// TwinCAT 3 PLC project Robotic
// ProgramVersion: 3.1.4023.0
// libraries:
//   CmpBitmapPool, * (System)
//   VisuElemMeter, * (System)
//   Tc2_EtherCAT, * (Beckhoff Automation GmbH)
//   Tc2_Standard, * (Beckhoff Automation GmbH)
//   Tc2_SUPS, * (Beckhoff Automation GmbH)
//   Tc2_System, * (Beckhoff Automation GmbH)
//   Tc2_Utilities, * (Beckhoff Automation GmbH)
//   Tc3_Module, * (Beckhoff Automation GmbH)
//   VisuDialogs, * (System)
//   VisuSymbols,3.5.10.0,System
//   VLT_ECAT_LIB_V1_12,1.12,Danfoss Drives
// project tree:
//   DUTs/OEE/ ShiftTime.TcDUT, Precentage_Time.TcDUT, ShiftCounter.TcDUT, sOEECounter.TcDUT, StartShift_EndShift.TcDUT, sOEETime.TcDUT
//   DUTs/Robot/ stCustomPattern.TcDUT, stProductInfo.TcDUT, stRobot_Input.TcDUT, stRobot_Output.TcDUT, unMyINT.TcDUT, unMyUINT.TcDUT
//   DUTs/ stCheckShuttle.TcDUT, stDM_Input.TcDUT, stDM_Output.TcDUT, stEcSlaveState.TcDUT, stErrorData.TcDUT, stMachineState.TcDUT, stMotor.TcDUT, stPalletTrackingData.TcDUT, stPneumatic1.TcDUT, stPneumatic2.TcDUT, stRejectData.TcDUT, stRTC_Data.TcDUT, stShuttle.TcDUT, stDataPallet.TcDUT
//   / Ethernet_Task.TcTTO, GlobalTextList.TcGTLO, IO_Task.TcTTO, Main_Task.TcTTO, Monitoring_Task.TcTTO, VISU_TASK.TcTTO
//   GVLs/ Data_GVL.TcGVL, HMI_GVL.TcGVL, InputOutput_GVL.TcGVL, Status_GVL.TcGVL
//   POUs/Function/ ConvertMilliSecTimeData.TcPOU, ConvertTimeToString.TcPOU
//   POUs/Function_Block/ FB_CheckShuttlePos.TcPOU
//   POUs/Function_Block/General/ Alarm_Event_History.TcPOU, Alarm_Event_Active.TcPOU, BLINK.TcPOU, CheckStatus.TcPOU, Ethercat_Status.TcPOU, FB_StateManager.TcPOU, FGHS_DataCollect_Palletizing.TcPOU, MotorManagement.TcPOU, OEETime.TcPOU, OEECounter.TcPOU, Pneumatic_1Coil_Management.TcPOU, Pneumatic_2Coil_Management.TcPOU, RejectMsgHandling.TcPOU, RTCManagement.TcPOU, SystemData.TcPOU
//   POUs/Function_Block/Placing/ FB_CustomOffset.TcPOU, FB_Placing.TcPOU, FB_Placing_v2.TcPOU, PalletID_Name.TcPOU
//   POUs/Function_Block/Robot/ DM_Connect.TcPOU, FB_BarcodeInspection.TcPOU, FB_Picking.TcPOU, FB_Recipe.TcPOU, RobotCustomPattern.TcPOU, FB_StartUpRobot.TcPOU, FB_Layer.TcPOU, RotatePick.TcPOU
//   POUs/S00_System_Utilities/ Backbone.TcPOU, IO_Mapping.TcPOU, Module_Status.TcPOU
//   POUs/S01_Robot/ EM01_Robot.TcPOU, EM06_Picking.TcPOU
//   POUs/S02_Placing/ EM02_Placing1.TcPOU, EM03_Placing2.TcPOU, EM04_Placing3.TcPOU, EM05_Placing4.TcPOU
//   VISUs/FGHS/ DataPallet2.TcVIS, DataPallet3.TcVIS, DataPallet4.TcVIS, FGHS.TcVIS, FGHS_1.TcVIS, DataPallet1.TcVIS
//   VISUs/Images/ ImagePool.TcIPO (not stored)
//   VISUs/Main/Alarm/ RejectMsg.TcVIS, AlarmHistory.TcVIS, AlarmActive.TcVIS, Alarm.TcVIS, PUDetail.TcVIS
//   VISUs/Main/ Header.TcVIS, Home.TcVIS, MainPage.TcVIS, Parameter.TcVIS, PLC_Status.TcVIS, PUSeq.TcVIS, StateMachine.TcVIS
//   VISUs/MTBF/ MTBF.TcVIS, MTBF_Picking.TcVIS, MTBF_Placing.TcVIS, MTBF_Outfeed.TcVIS, MTBF_Infeed.TcVIS, MTBF_Shuttle.TcVIS, MTBF_Dispenser.TcVIS
//   VISUs/OEE/ OEE.TcVIS, OEE_Outfeed.TcVIS, OEE_Robot.TcVIS, OEE_Counter.TcVIS
//   VISUs/Parameter/ LinkUp.TcTLO, MShuttle.TcVIS, MOutfeed.TcVIS, MInfeed.TcVIS, MDispenser.TcVIS, MPicking.TcVIS, MPlacing.TcVIS
//   VISUs/Parameter/Recipe/ MOffset_2.TcVIS, MOffset_3.TcVIS, MOffset_4.TcVIS, MRecipe.TcVIS, MRecipe_1.TcVIS, MOffset_1.TcVIS, MRecipe_2.TcVIS, MRecipe_3.TcVIS, MRecipe_4.TcVIS
//   VISUs/PLC Status/P1 - Panel Robot/ P1_DI1.TcVIS, P1_DI2.TcVIS, P1_DI3.TcVIS, P1_DI4.TcVIS, P1_DO1.TcVIS, P1_DO2.TcVIS, P1_DO3.TcVIS
//   VISUs/PLC Status/P2 - Panel Outfeed/ P2_DI1.TcVIS, P2_DI2.TcVIS, P2_DI3.TcVIS, P2_DI4.TcVIS, P2_DI5.TcVIS, P2_DI6.TcVIS, P2_DI7.TcVIS, P2_DO1.TcVIS, P2_DO2.TcVIS, P2_DO3.TcVIS, P2_DO4.TcVIS
//   VISUs/PLC Status/P3 - Panel Shuttle/ P3_DI1.TcVIS, P3_DO1.TcVIS
//   VISUs/PLC Status/ SeqStatus.TcVIS, IO_Status.TcVIS
//   VISUs/TestMode/ Test_Outfeed.TcVIS, Control.TcVIS, Test_Infeed.TcVIS, Test_Place1.TcVIS, Test_Place2.TcVIS, Test_Place3.TcVIS, Test_Place4.TcVIS, Test_Shuttle.TcVIS, Test_Picking.TcVIS
//   VISUs/ VisualizationManager.TcVMO (not stored)
// real-time tasks:
//   TASK Main_Task: cycle T#4ms, priority 2, ADS port 350
//   TASK IO_Task: cycle T#2ms, priority 1, ADS port 351
//   TASK Monitoring_Task: cycle T#10ms, priority 10, ADS port 352
//   TASK Ethernet_Task: cycle T#100000us, priority 3, ADS port 353
//   TASK VISU_TASK: cycle T#100000us, priority 30, ADS port 354
// I/O:
//   DEVICE Main Panel (EtherCAT), AmsNetId 5.104.237.244.2.1
//     Term 1 (EK1200) [EK1200-5000 EtherCAT Power supply (2A E-Bus)]
//       Term 2 (EL1809) [EL1809 16Ch. Dig. Input 24V, 3ms]
//       Term 3 (EL1809) [EL1809 16Ch. Dig. Input 24V, 3ms]
//       Term 4 (EL1809) [EL1809 16Ch. Dig. Input 24V, 3ms]
//       Term 5 (EL1809) [EL1809 16Ch. Dig. Input 24V, 3ms]
//       Term 6 (EL2809) [EL2809 16Ch. Dig. Output 24V, 0.5A]
//       Term 7 (EL2809) [EL2809 16Ch. Dig. Output 24V, 0.5A]
//       Term 8 (EL2809) [EL2809 16Ch. Dig. Output 24V, 0.5A]
//       DeviceNet Master (EL6752) [EL6752 DeviceNet Master]
//   DEVICE Device 2 (EL6752), AmsNetId 5.104.237.244.3.1
//     Box 10 (Robot) // EDS-File: 'IRC5_Slave_DSQC1006.eds' DescText: Molex SST-DN4 Scanner EDS File Vendor: Molex Software & Electronics (SST) Device Type: Communication Adapter Product Name: Molex SST-DN4 Scanner Catalog Number: 0
//   DEVICE Ethernet/IP, AmsNetId 5.104.237.244.4.1
//     Box 11 (DataMan 300 Series Reader) // <INFO> </INFO> <EDS> C:\TwinCAT\3.1\Config\Io\EtherNetIP\0678077312900100.eds </EDS>
//     Box 12 (DataMan 260 Series Reader) (disabled) // <INFO> </INFO> <EDS> C:\TwinCAT\3.1\Config\Io\EtherNetIP\0678077313070100.eds </EDS>
//     Box 13 (DataMan 260 Series Reader) (disabled) // <INFO> </INFO> <EDS> C:\TwinCAT\3.1\Config\Io\EtherNetIP\0678077313070100.eds </EDS>
//     Box 14 (DataMan 300 Series Reader) // <INFO> </INFO> <EDS> C:\TwinCAT\3.1\Config\Io\EtherNetIP\0678077312900100.eds </EDS>
//     Box 17 (DataMan DM280) // <INFO> </INFO> <EDS> C:\TwinCAT\3.1\Config\Io\EtherNetIP\02A60305052E0100.eds </EDS>
//     Box 18 (DataMan 300 Series Reader) // <INFO> </INFO> <EDS> C:\TwinCAT\3.1\Config\Io\EtherNetIP\0678077312900100.eds </EDS>
//   DEVICE Device 4 (EtherCAT Automation Protocol), AmsNetId 5.104.237.244.5.1
//     Box 15 (Publisher)
//     Box 16 (Subscriber)
// variable links:
//   Robotic/Robotic Instance <-> Device 2 (EL6752)/Box 10 (Robot)
//     IO_Task Inputs/InputOutput_GVL.xIn_ConnectionRobot[{1..64}] <-> Connection (Poll)/Inputs/In_{1..64}  (64 links)
//     IO_Task Outputs/InputOutput_GVL.xOut_ConnectionRobot[{1..64}] <-> Connection (Poll)/Outputs/Out_{1..64}  (64 links)
//   Robotic/Robotic Instance <-> Device 4 (EtherCAT Automation Protocol)/Box 15 (Publisher)
//     Main_Task Outputs/InputOutput_GVL.ControlButton <-> ControlButton/Outputs/VarData
//     Main_Task Outputs/InputOutput_GVL.Counter <-> Counter/Outputs/VarData
//     Main_Task Outputs/InputOutput_GVL.PickingBusy <-> PickingBusy/Outputs/VarData
//     Main_Task Outputs/InputOutput_GVL.RequestEmptyPallet <-> ReqEmpty/Outputs/VarData
//     Main_Task Outputs/InputOutput_GVL.RequestLoadPallet <-> ReqLoad/Outputs/VarData
//     Main_Task Outputs/InputOutput_GVL.Shuttle_Offset <-> Shuttle_Offset/Outputs/VarData
//     Main_Task Outputs/InputOutput_GVL.Shuttle_Speed <-> Shuttle_Speed/Outputs/VarData
//     Main_Task Outputs/InputOutput_GVL.TestMode <-> TestMode/Outputs/VarData
//     Main_Task Outputs/InputOutput_GVL.TmrOutfeed <-> TmrOutfeed/Outputs/VarData
//     Main_Task Outputs/InputOutput_GVL.stShuttleSequence <-> stShuttleSequence/Outputs/VarData
//     Monitoring_Task Outputs/InputOutput_GVL.Error_Safety <-> Error_Safety/Outputs/VarData
//   Robotic/Robotic Instance <-> Device 4 (EtherCAT Automation Protocol)/Box 16 (Subscriber)
//     Main_Task Inputs/InputOutput_GVL.Digital_Output <-> Digital_Output/Inputs/VarData
//     Main_Task Inputs/InputOutput_GVL.ErrorShuttleEmpty <-> ErrorShuttleEmpty/Inputs/VarData
//     Main_Task Inputs/InputOutput_GVL.ErrorShuttleLoad <-> ErrorShuttleLoad/Inputs/VarData
//     Main_Task Inputs/InputOutput_GVL.FB_RequestShuttle <-> FB_RequestShuttle/Inputs/VarData
//     Main_Task Inputs/InputOutput_GVL.Infeed_stsMachine <-> Infeed_stsMachine/Inputs/VarData
//     Main_Task Inputs/InputOutput_GVL.LoadPalletGoOut <-> LoadPalletGoOut/Inputs/VarData
//     Main_Task Inputs/InputOutput_GVL.Outfeed_stsMachine <-> Outfeed_stsMachine/Inputs/VarData
//     Main_Task Inputs/InputOutput_GVL.SeqIndexOutfeed <-> SeqIndex/Inputs/VarData
//     Main_Task Inputs/InputOutput_GVL.ShuttlePosition <-> ShuttlePos/Inputs/VarData
//     Main_Task Inputs/InputOutput_GVL.Shuttle_stsMachine <-> Shuttle_stsMachine/Inputs/VarData
//     Main_Task Inputs/InputOutput_GVL.stErrorDispenser <-> stErrorDispenser/Inputs/VarData
//     Main_Task Inputs/InputOutput_GVL.stErrorInfeed <-> stErrorInfeed/Inputs/VarData
//     Main_Task Inputs/InputOutput_GVL.stErrorOutfeed <-> stErrorOutfeed/Inputs/VarData
//     Main_Task Inputs/InputOutput_GVL.stErrorShuttle <-> stErrorShuttle/Inputs/VarData
//     Monitoring_Task Inputs/InputOutput_GVL.Digital_Input <-> Digital_Input/Inputs/VarData
//     Monitoring_Task Inputs/InputOutput_GVL.Dispenser_stsMachine <-> Dispenser_stsMachine/Inputs/VarData
//     Monitoring_Task Inputs/InputOutput_GVL.MTBF_Motor <-> MTBF_Motor/Inputs/VarData
//     Monitoring_Task Inputs/InputOutput_GVL.MTBF_Pneumatic <-> MTBF_Pneumatic/Inputs/VarData
//   Robotic/Robotic Instance <-> Ethernet/IP/Box 11 (DataMan 300 Series Reader)
//     Main_Task Inputs/InputOutput_GVL.xIn_BarcodeReader_Picking1/Acquiring <-> Connection 1 (Input/Output)/Inputs/Acquiring
//     Main_Task Inputs/InputOutput_GVL.xIn_BarcodeReader_Picking1/DecodeComplete <-> Connection 1 (Input/Output)/Inputs/Decode Complete
//     Main_Task Inputs/InputOutput_GVL.xIn_BarcodeReader_Picking1/Decoding <-> Connection 1 (Input/Output)/Inputs/Decoding
//     Main_Task Inputs/InputOutput_GVL.xIn_BarcodeReader_Picking1/GeneralFault <-> Connection 1 (Input/Output)/Inputs/General Fault
//     Main_Task Inputs/InputOutput_GVL.xIn_BarcodeReader_Picking1/MissedAcq <-> Connection 1 (Input/Output)/Inputs/Missed Acq
//     Main_Task Inputs/InputOutput_GVL.xIn_BarcodeReader_Picking1/ResultCode <-> Connection 1 (Input/Output)/Inputs/Result Code
//     Main_Task Inputs/InputOutput_GVL.xIn_BarcodeReader_Picking1/ResultData <-> Connection 1 (Input/Output)/Inputs/ResultData
//     Main_Task Inputs/InputOutput_GVL.xIn_BarcodeReader_Picking1/ResultDataLength <-> Connection 1 (Input/Output)/Inputs/Result Length
//     Main_Task Inputs/InputOutput_GVL.xIn_BarcodeReader_Picking1/ResultExtended <-> Connection 1 (Input/Output)/Inputs/Result Extended
//     Main_Task Inputs/InputOutput_GVL.xIn_BarcodeReader_Picking1/ResultID <-> Connection 1 (Input/Output)/Inputs/Result ID
//     Main_Task Inputs/InputOutput_GVL.xIn_BarcodeReader_Picking1/ResultsAvailable <-> Connection 1 (Input/Output)/Inputs/Results Available
//     Main_Task Inputs/InputOutput_GVL.xIn_BarcodeReader_Picking1/ResultsBufferOverrun <-> Connection 1 (Input/Output)/Inputs/Results Buffer Overrun
//     Main_Task Inputs/InputOutput_GVL.xIn_BarcodeReader_Picking1/TriggerAck <-> Connection 1 (Input/Output)/Inputs/Trigger Ack
//     Main_Task Inputs/InputOutput_GVL.xIn_BarcodeReader_Picking1/TriggerID <-> Connection 1 (Input/Output)/Inputs/Trigger ID
//     Main_Task Inputs/InputOutput_GVL.xIn_BarcodeReader_Picking1/TriggerReady <-> Connection 1 (Input/Output)/Inputs/Trigger Ready
//     Main_Task Outputs/InputOutput_GVL.xOut_BarcodeReader_Picking1/BufferResultsEnable <-> Connection 1 (Input/Output)/Outputs/Buffer Results Enable
//     Main_Task Outputs/InputOutput_GVL.xOut_BarcodeReader_Picking1/ResultsAck <-> Connection 1 (Input/Output)/Outputs/Results Ack
//     Main_Task Outputs/InputOutput_GVL.xOut_BarcodeReader_Picking1/Trigger <-> Connection 1 (Input/Output)/Outputs/Trigger
//     Main_Task Outputs/InputOutput_GVL.xOut_BarcodeReader_Picking1/TriggerEnable <-> Connection 1 (Input/Output)/Outputs/Trigger Enable
//     Main_Task Outputs/InputOutput_GVL.xOut_BarcodeReader_Picking1/UserData <-> Connection 1 (Input/Output)/Outputs/UserData
//     Main_Task Outputs/InputOutput_GVL.xOut_BarcodeReader_Picking1/UserDataLength <-> Connection 1 (Input/Output)/Outputs/User Data Length
//     Main_Task Outputs/InputOutput_GVL.xOut_BarcodeReader_Picking1/UserDataOption <-> Connection 1 (Input/Output)/Outputs/User Data Option
//     Monitoring_Task Inputs/InputOutput_GVL.BarcodeReader_Picking1_State <-> Inputs/State
//   Robotic/Robotic Instance <-> Ethernet/IP/Box 12 (DataMan 260 Series Reader)
//     Monitoring_Task Inputs/InputOutput_GVL.BarcodeReader_Picking2_State <-> Inputs/State
//     Monitoring_Task Inputs/InputOutput_GVL.xIn_BarcodeReader_Picking2/Acquiring <-> Connection 2 (Input/Output)/Inputs/Acquiring
//     Monitoring_Task Inputs/InputOutput_GVL.xIn_BarcodeReader_Picking2/DecodeComplete <-> Connection 2 (Input/Output)/Inputs/Decode Complete
//     Monitoring_Task Inputs/InputOutput_GVL.xIn_BarcodeReader_Picking2/Decoding <-> Connection 2 (Input/Output)/Inputs/Decoding
//     Monitoring_Task Inputs/InputOutput_GVL.xIn_BarcodeReader_Picking2/GeneralFault <-> Connection 2 (Input/Output)/Inputs/General Fault
//     Monitoring_Task Inputs/InputOutput_GVL.xIn_BarcodeReader_Picking2/MissedAcq <-> Connection 2 (Input/Output)/Inputs/Missed Acq
//     Monitoring_Task Inputs/InputOutput_GVL.xIn_BarcodeReader_Picking2/ResultCode <-> Connection 2 (Input/Output)/Inputs/Result Code
//     Monitoring_Task Inputs/InputOutput_GVL.xIn_BarcodeReader_Picking2/ResultData <-> Connection 2 (Input/Output)/Inputs/ResultData
//     Monitoring_Task Inputs/InputOutput_GVL.xIn_BarcodeReader_Picking2/ResultDataLength <-> Connection 2 (Input/Output)/Inputs/Result Length
//     Monitoring_Task Inputs/InputOutput_GVL.xIn_BarcodeReader_Picking2/ResultExtended <-> Connection 2 (Input/Output)/Inputs/Result Extended
//     Monitoring_Task Inputs/InputOutput_GVL.xIn_BarcodeReader_Picking2/ResultID <-> Connection 2 (Input/Output)/Inputs/Result ID
//     Monitoring_Task Inputs/InputOutput_GVL.xIn_BarcodeReader_Picking2/ResultsAvailable <-> Connection 2 (Input/Output)/Inputs/Results Available
//     Monitoring_Task Inputs/InputOutput_GVL.xIn_BarcodeReader_Picking2/ResultsBufferOverrun <-> Connection 2 (Input/Output)/Inputs/Results Buffer Overrun
//     Monitoring_Task Inputs/InputOutput_GVL.xIn_BarcodeReader_Picking2/TriggerAck <-> Connection 2 (Input/Output)/Inputs/Trigger Ack
//     Monitoring_Task Inputs/InputOutput_GVL.xIn_BarcodeReader_Picking2/TriggerID <-> Connection 2 (Input/Output)/Inputs/Trigger ID
//     Monitoring_Task Inputs/InputOutput_GVL.xIn_BarcodeReader_Picking2/TriggerReady <-> Connection 2 (Input/Output)/Inputs/Trigger Ready
//     Monitoring_Task Outputs/InputOutput_GVL.xOut_BarcodeReader_Picking2/BufferResultsEnable <-> Connection 2 (Input/Output)/Outputs/Buffer Results Enable
//     Monitoring_Task Outputs/InputOutput_GVL.xOut_BarcodeReader_Picking2/ResultsAck <-> Connection 2 (Input/Output)/Outputs/Results Ack
//     Monitoring_Task Outputs/InputOutput_GVL.xOut_BarcodeReader_Picking2/Trigger <-> Connection 2 (Input/Output)/Outputs/Trigger
//     Monitoring_Task Outputs/InputOutput_GVL.xOut_BarcodeReader_Picking2/TriggerEnable <-> Connection 2 (Input/Output)/Outputs/Trigger Enable
//     Monitoring_Task Outputs/InputOutput_GVL.xOut_BarcodeReader_Picking2/UserData <-> Connection 2 (Input/Output)/Outputs/UserData
//     Monitoring_Task Outputs/InputOutput_GVL.xOut_BarcodeReader_Picking2/UserDataLength <-> Connection 2 (Input/Output)/Outputs/User Data Length
//     Monitoring_Task Outputs/InputOutput_GVL.xOut_BarcodeReader_Picking2/UserDataOption <-> Connection 2 (Input/Output)/Outputs/User Data Option
//   Robotic/Robotic Instance <-> Ethernet/IP/Box 13 (DataMan 260 Series Reader)
//     Monitoring_Task Inputs/InputOutput_GVL.BarcodeReader_Picking3_State <-> Inputs/State
//     Monitoring_Task Inputs/InputOutput_GVL.xIn_BarcodeReader_Picking3/Acquiring <-> Connection 3 (Input/Output)/Inputs/Acquiring
//     Monitoring_Task Inputs/InputOutput_GVL.xIn_BarcodeReader_Picking3/DecodeComplete <-> Connection 3 (Input/Output)/Inputs/Decode Complete
//     Monitoring_Task Inputs/InputOutput_GVL.xIn_BarcodeReader_Picking3/Decoding <-> Connection 3 (Input/Output)/Inputs/Decoding
//     Monitoring_Task Inputs/InputOutput_GVL.xIn_BarcodeReader_Picking3/GeneralFault <-> Connection 3 (Input/Output)/Inputs/General Fault
//     Monitoring_Task Inputs/InputOutput_GVL.xIn_BarcodeReader_Picking3/MissedAcq <-> Connection 3 (Input/Output)/Inputs/Missed Acq
//     Monitoring_Task Inputs/InputOutput_GVL.xIn_BarcodeReader_Picking3/ResultCode <-> Connection 3 (Input/Output)/Inputs/Result Code
//     Monitoring_Task Inputs/InputOutput_GVL.xIn_BarcodeReader_Picking3/ResultData <-> Connection 3 (Input/Output)/Inputs/ResultData
//     Monitoring_Task Inputs/InputOutput_GVL.xIn_BarcodeReader_Picking3/ResultDataLength <-> Connection 3 (Input/Output)/Inputs/Result Length
//     Monitoring_Task Inputs/InputOutput_GVL.xIn_BarcodeReader_Picking3/ResultExtended <-> Connection 3 (Input/Output)/Inputs/Result Extended
//     Monitoring_Task Inputs/InputOutput_GVL.xIn_BarcodeReader_Picking3/ResultID <-> Connection 3 (Input/Output)/Inputs/Result ID
//     Monitoring_Task Inputs/InputOutput_GVL.xIn_BarcodeReader_Picking3/ResultsAvailable <-> Connection 3 (Input/Output)/Inputs/Results Available
//     Monitoring_Task Inputs/InputOutput_GVL.xIn_BarcodeReader_Picking3/ResultsBufferOverrun <-> Connection 3 (Input/Output)/Inputs/Results Buffer Overrun
//     Monitoring_Task Inputs/InputOutput_GVL.xIn_BarcodeReader_Picking3/TriggerAck <-> Connection 3 (Input/Output)/Inputs/Trigger Ack
//     Monitoring_Task Inputs/InputOutput_GVL.xIn_BarcodeReader_Picking3/TriggerID <-> Connection 3 (Input/Output)/Inputs/Trigger ID
//     Monitoring_Task Inputs/InputOutput_GVL.xIn_BarcodeReader_Picking3/TriggerReady <-> Connection 3 (Input/Output)/Inputs/Trigger Ready
//     Monitoring_Task Outputs/InputOutput_GVL.xOut_BarcodeReader_Picking3/BufferResultsEnable <-> Connection 3 (Input/Output)/Outputs/Buffer Results Enable
//     Monitoring_Task Outputs/InputOutput_GVL.xOut_BarcodeReader_Picking3/ResultsAck <-> Connection 3 (Input/Output)/Outputs/Results Ack
//     Monitoring_Task Outputs/InputOutput_GVL.xOut_BarcodeReader_Picking3/Trigger <-> Connection 3 (Input/Output)/Outputs/Trigger
//     Monitoring_Task Outputs/InputOutput_GVL.xOut_BarcodeReader_Picking3/TriggerEnable <-> Connection 3 (Input/Output)/Outputs/Trigger Enable
//     Monitoring_Task Outputs/InputOutput_GVL.xOut_BarcodeReader_Picking3/UserData <-> Connection 3 (Input/Output)/Outputs/UserData
//     Monitoring_Task Outputs/InputOutput_GVL.xOut_BarcodeReader_Picking3/UserDataLength <-> Connection 3 (Input/Output)/Outputs/User Data Length
//     Monitoring_Task Outputs/InputOutput_GVL.xOut_BarcodeReader_Picking3/UserDataOption <-> Connection 3 (Input/Output)/Outputs/User Data Option
//   Robotic/Robotic Instance <-> Ethernet/IP/Box 14 (DataMan 300 Series Reader)
//     Main_Task Inputs/InputOutput_GVL.xIn_BarcodeReader_Picking4/Acquiring <-> Connection 4 (Input/Output)/Inputs/Acquiring
//     Main_Task Inputs/InputOutput_GVL.xIn_BarcodeReader_Picking4/DecodeComplete <-> Connection 4 (Input/Output)/Inputs/Decode Complete
//     Main_Task Inputs/InputOutput_GVL.xIn_BarcodeReader_Picking4/Decoding <-> Connection 4 (Input/Output)/Inputs/Decoding
//     Main_Task Inputs/InputOutput_GVL.xIn_BarcodeReader_Picking4/GeneralFault <-> Connection 4 (Input/Output)/Inputs/General Fault
//     Main_Task Inputs/InputOutput_GVL.xIn_BarcodeReader_Picking4/MissedAcq <-> Connection 4 (Input/Output)/Inputs/Missed Acq
//     Main_Task Inputs/InputOutput_GVL.xIn_BarcodeReader_Picking4/ResultCode <-> Connection 4 (Input/Output)/Inputs/Result Code
//     Main_Task Inputs/InputOutput_GVL.xIn_BarcodeReader_Picking4/ResultData <-> Connection 4 (Input/Output)/Inputs/ResultData
//     Main_Task Inputs/InputOutput_GVL.xIn_BarcodeReader_Picking4/ResultDataLength <-> Connection 4 (Input/Output)/Inputs/Result Length
//     Main_Task Inputs/InputOutput_GVL.xIn_BarcodeReader_Picking4/ResultExtended <-> Connection 4 (Input/Output)/Inputs/Result Extended
//     Main_Task Inputs/InputOutput_GVL.xIn_BarcodeReader_Picking4/ResultID <-> Connection 4 (Input/Output)/Inputs/Result ID
//     Main_Task Inputs/InputOutput_GVL.xIn_BarcodeReader_Picking4/ResultsAvailable <-> Connection 4 (Input/Output)/Inputs/Results Available
//     Main_Task Inputs/InputOutput_GVL.xIn_BarcodeReader_Picking4/ResultsBufferOverrun <-> Connection 4 (Input/Output)/Inputs/Results Buffer Overrun
//     Main_Task Inputs/InputOutput_GVL.xIn_BarcodeReader_Picking4/TriggerAck <-> Connection 4 (Input/Output)/Inputs/Trigger Ack
//     Main_Task Inputs/InputOutput_GVL.xIn_BarcodeReader_Picking4/TriggerID <-> Connection 4 (Input/Output)/Inputs/Trigger ID
//     Main_Task Inputs/InputOutput_GVL.xIn_BarcodeReader_Picking4/TriggerReady <-> Connection 4 (Input/Output)/Inputs/Trigger Ready
//     Main_Task Outputs/InputOutput_GVL.xOut_BarcodeReader_Picking4/BufferResultsEnable <-> Connection 4 (Input/Output)/Outputs/Buffer Results Enable
//     Main_Task Outputs/InputOutput_GVL.xOut_BarcodeReader_Picking4/ResultsAck <-> Connection 4 (Input/Output)/Outputs/Results Ack
//     Main_Task Outputs/InputOutput_GVL.xOut_BarcodeReader_Picking4/Trigger <-> Connection 4 (Input/Output)/Outputs/Trigger
//     Main_Task Outputs/InputOutput_GVL.xOut_BarcodeReader_Picking4/TriggerEnable <-> Connection 4 (Input/Output)/Outputs/Trigger Enable
//     Main_Task Outputs/InputOutput_GVL.xOut_BarcodeReader_Picking4/UserData <-> Connection 4 (Input/Output)/Outputs/UserData
//     Main_Task Outputs/InputOutput_GVL.xOut_BarcodeReader_Picking4/UserDataLength <-> Connection 4 (Input/Output)/Outputs/User Data Length
//     Main_Task Outputs/InputOutput_GVL.xOut_BarcodeReader_Picking4/UserDataOption <-> Connection 4 (Input/Output)/Outputs/User Data Option
//     Monitoring_Task Inputs/InputOutput_GVL.BarcodeReader_Picking4_State <-> Inputs/State
//   Robotic/Robotic Instance <-> Ethernet/IP/Box 17 (DataMan DM280)
//     Main_Task Inputs/InputOutput_GVL.xIn_BarcodeReader_Picking2B/Acquiring <-> Connection 5 (Input/Output)/Inputs/Acquiring
//     Main_Task Inputs/InputOutput_GVL.xIn_BarcodeReader_Picking2B/DecodeComplete <-> Connection 5 (Input/Output)/Inputs/Decode Complete
//     Main_Task Inputs/InputOutput_GVL.xIn_BarcodeReader_Picking2B/Decoding <-> Connection 5 (Input/Output)/Inputs/Decoding
//     Main_Task Inputs/InputOutput_GVL.xIn_BarcodeReader_Picking2B/GeneralFault <-> Connection 5 (Input/Output)/Inputs/General Fault
//     Main_Task Inputs/InputOutput_GVL.xIn_BarcodeReader_Picking2B/MissedAcq <-> Connection 5 (Input/Output)/Inputs/Missed Acq
//     Main_Task Inputs/InputOutput_GVL.xIn_BarcodeReader_Picking2B/ResultCode <-> Connection 5 (Input/Output)/Inputs/Result Code
//     Main_Task Inputs/InputOutput_GVL.xIn_BarcodeReader_Picking2B/ResultData <-> Connection 5 (Input/Output)/Inputs/ResultData
//     Main_Task Inputs/InputOutput_GVL.xIn_BarcodeReader_Picking2B/ResultDataLength <-> Connection 5 (Input/Output)/Inputs/Result Length
//     Main_Task Inputs/InputOutput_GVL.xIn_BarcodeReader_Picking2B/ResultExtended <-> Connection 5 (Input/Output)/Inputs/Result Extended
//     Main_Task Inputs/InputOutput_GVL.xIn_BarcodeReader_Picking2B/ResultID <-> Connection 5 (Input/Output)/Inputs/Result ID
//     Main_Task Inputs/InputOutput_GVL.xIn_BarcodeReader_Picking2B/ResultsAvailable <-> Connection 5 (Input/Output)/Inputs/Results Available
//     Main_Task Inputs/InputOutput_GVL.xIn_BarcodeReader_Picking2B/ResultsBufferOverrun <-> Connection 5 (Input/Output)/Inputs/Results Buffer Overrun
//     Main_Task Inputs/InputOutput_GVL.xIn_BarcodeReader_Picking2B/TriggerAck <-> Connection 5 (Input/Output)/Inputs/Trigger Ack
//     Main_Task Inputs/InputOutput_GVL.xIn_BarcodeReader_Picking2B/TriggerID <-> Connection 5 (Input/Output)/Inputs/Trigger ID
//     Main_Task Inputs/InputOutput_GVL.xIn_BarcodeReader_Picking2B/TriggerReady <-> Connection 5 (Input/Output)/Inputs/Trigger Ready
//     Main_Task Outputs/InputOutput_GVL.xOut_BarcodeReader_Picking2B/BufferResultsEnable <-> Connection 5 (Input/Output)/Outputs/Buffer Results Enable
//     Main_Task Outputs/InputOutput_GVL.xOut_BarcodeReader_Picking2B/ResultsAck <-> Connection 5 (Input/Output)/Outputs/Results Ack
//     Main_Task Outputs/InputOutput_GVL.xOut_BarcodeReader_Picking2B/Trigger <-> Connection 5 (Input/Output)/Outputs/Trigger
//     Main_Task Outputs/InputOutput_GVL.xOut_BarcodeReader_Picking2B/TriggerEnable <-> Connection 5 (Input/Output)/Outputs/Trigger Enable
//     Main_Task Outputs/InputOutput_GVL.xOut_BarcodeReader_Picking2B/UserData <-> Connection 5 (Input/Output)/Outputs/UserData
//     Main_Task Outputs/InputOutput_GVL.xOut_BarcodeReader_Picking2B/UserDataLength <-> Connection 5 (Input/Output)/Outputs/User Data Length
//     Main_Task Outputs/InputOutput_GVL.xOut_BarcodeReader_Picking2B/UserDataOption <-> Connection 5 (Input/Output)/Outputs/User Data Option
//     Monitoring_Task Inputs/InputOutput_GVL.BarcodeReader_Picking2B_State <-> Inputs/State
//   Robotic/Robotic Instance <-> Ethernet/IP/Box 18 (DataMan 300 Series Reader)
//     Main_Task Inputs/InputOutput_GVL.xIn_BarcodeReader_Picking3B/Acquiring <-> Connection 6 (Input/Output)/Inputs/Acquiring
//     Main_Task Inputs/InputOutput_GVL.xIn_BarcodeReader_Picking3B/DecodeComplete <-> Connection 6 (Input/Output)/Inputs/Decode Complete
//     Main_Task Inputs/InputOutput_GVL.xIn_BarcodeReader_Picking3B/Decoding <-> Connection 6 (Input/Output)/Inputs/Decoding
//     Main_Task Inputs/InputOutput_GVL.xIn_BarcodeReader_Picking3B/GeneralFault <-> Connection 6 (Input/Output)/Inputs/General Fault
//     Main_Task Inputs/InputOutput_GVL.xIn_BarcodeReader_Picking3B/MissedAcq <-> Connection 6 (Input/Output)/Inputs/Missed Acq
//     Main_Task Inputs/InputOutput_GVL.xIn_BarcodeReader_Picking3B/ResultCode <-> Connection 6 (Input/Output)/Inputs/Result Code
//     Main_Task Inputs/InputOutput_GVL.xIn_BarcodeReader_Picking3B/ResultData <-> Connection 6 (Input/Output)/Inputs/ResultData
//     Main_Task Inputs/InputOutput_GVL.xIn_BarcodeReader_Picking3B/ResultDataLength <-> Connection 6 (Input/Output)/Inputs/Result Length
//     Main_Task Inputs/InputOutput_GVL.xIn_BarcodeReader_Picking3B/ResultExtended <-> Connection 6 (Input/Output)/Inputs/Result Extended
//     Main_Task Inputs/InputOutput_GVL.xIn_BarcodeReader_Picking3B/ResultID <-> Connection 6 (Input/Output)/Inputs/Result ID
//     Main_Task Inputs/InputOutput_GVL.xIn_BarcodeReader_Picking3B/ResultsAvailable <-> Connection 6 (Input/Output)/Inputs/Results Available
//     Main_Task Inputs/InputOutput_GVL.xIn_BarcodeReader_Picking3B/ResultsBufferOverrun <-> Connection 6 (Input/Output)/Inputs/Results Buffer Overrun
//     Main_Task Inputs/InputOutput_GVL.xIn_BarcodeReader_Picking3B/TriggerAck <-> Connection 6 (Input/Output)/Inputs/Trigger Ack
//     Main_Task Inputs/InputOutput_GVL.xIn_BarcodeReader_Picking3B/TriggerID <-> Connection 6 (Input/Output)/Inputs/Trigger ID
//     Main_Task Inputs/InputOutput_GVL.xIn_BarcodeReader_Picking3B/TriggerReady <-> Connection 6 (Input/Output)/Inputs/Trigger Ready
//     Main_Task Outputs/InputOutput_GVL.xOut_BarcodeReader_Picking3B/BufferResultsEnable <-> Connection 6 (Input/Output)/Outputs/Buffer Results Enable
//     Main_Task Outputs/InputOutput_GVL.xOut_BarcodeReader_Picking3B/ResultsAck <-> Connection 6 (Input/Output)/Outputs/Results Ack
//     Main_Task Outputs/InputOutput_GVL.xOut_BarcodeReader_Picking3B/Trigger <-> Connection 6 (Input/Output)/Outputs/Trigger
//     Main_Task Outputs/InputOutput_GVL.xOut_BarcodeReader_Picking3B/TriggerEnable <-> Connection 6 (Input/Output)/Outputs/Trigger Enable
//     Main_Task Outputs/InputOutput_GVL.xOut_BarcodeReader_Picking3B/UserData <-> Connection 6 (Input/Output)/Outputs/UserData
//     Main_Task Outputs/InputOutput_GVL.xOut_BarcodeReader_Picking3B/UserDataLength <-> Connection 6 (Input/Output)/Outputs/User Data Length
//     Main_Task Outputs/InputOutput_GVL.xOut_BarcodeReader_Picking3B/UserDataOption <-> Connection 6 (Input/Output)/Outputs/User Data Option
//     Monitoring_Task Inputs/InputOutput_GVL.BarcodeReader_Picking3B_State <-> Inputs/State
//   Robotic/Robotic Instance <-> Main Panel (EtherCAT)/Term 1 (EK1200)/Term 2 (EL1809)
//     IO_Task Inputs/InputOutput_GVL.xIn1000 <-> Channel 1/Input
//     IO_Task Inputs/InputOutput_GVL.xIn1001 <-> Channel 2/Input
//     IO_Task Inputs/InputOutput_GVL.xIn1002 <-> Channel 3/Input
//     IO_Task Inputs/InputOutput_GVL.xIn1003 <-> Channel 4/Input
//     IO_Task Inputs/InputOutput_GVL.xIn1004 <-> Channel 5/Input
//     IO_Task Inputs/InputOutput_GVL.xIn1005 <-> Channel 6/Input
//     IO_Task Inputs/InputOutput_GVL.xIn1015 <-> Channel 16/Input
//     Monitoring_Task Inputs/InputOutput_GVL.xIn{1006..1014} <-> Channel {7..15}/Input  (9 links)
//   Robotic/Robotic Instance <-> Main Panel (EtherCAT)/Term 1 (EK1200)/Term 3 (EL1809)
//     IO_Task Inputs/InputOutput_GVL.xIn1200 <-> Channel 1/Input
//     IO_Task Inputs/InputOutput_GVL.xIn1202 <-> Channel 3/Input
//     IO_Task Inputs/InputOutput_GVL.xIn1203 <-> Channel 4/Input
//     IO_Task Inputs/InputOutput_GVL.xIn1204 <-> Channel 5/Input
//     IO_Task Inputs/InputOutput_GVL.xIn1205 <-> Channel 6/Input
//     IO_Task Inputs/InputOutput_GVL.xIn1211 <-> Channel 12/Input
//     IO_Task Inputs/InputOutput_GVL.xIn1212 <-> Channel 13/Input
//     IO_Task Inputs/InputOutput_GVL.xIn1213 <-> Channel 14/Input
//     IO_Task Inputs/InputOutput_GVL.xIn1214 <-> Channel 15/Input
//     Monitoring_Task Inputs/InputOutput_GVL.xIn1201 <-> Channel 2/Input
//     Monitoring_Task Inputs/InputOutput_GVL.xIn1206 <-> Channel 7/Input
//     Monitoring_Task Inputs/InputOutput_GVL.xIn1207 <-> Channel 8/Input
//     Monitoring_Task Inputs/InputOutput_GVL.xIn1208 <-> Channel 9/Input
//     Monitoring_Task Inputs/InputOutput_GVL.xIn1209 <-> Channel 10/Input
//     Monitoring_Task Inputs/InputOutput_GVL.xIn1210 <-> Channel 11/Input
//     Monitoring_Task Inputs/InputOutput_GVL.xIn1215 <-> Channel 16/Input
//   Robotic/Robotic Instance <-> Main Panel (EtherCAT)/Term 1 (EK1200)/Term 4 (EL1809)
//     IO_Task Inputs/InputOutput_GVL.xIn1400 <-> Channel 1/Input
//     IO_Task Inputs/InputOutput_GVL.xIn1401 <-> Channel 2/Input
//     IO_Task Inputs/InputOutput_GVL.xIn1402 <-> Channel 3/Input
//     IO_Task Inputs/InputOutput_GVL.xIn1403 <-> Channel 4/Input
//     IO_Task Inputs/InputOutput_GVL.xIn1404 <-> Channel 5/Input
//     IO_Task Inputs/InputOutput_GVL.xIn1405 <-> Channel 6/Input
//     IO_Task Inputs/InputOutput_GVL.xIn1406 <-> Channel 7/Input
//     IO_Task Inputs/InputOutput_GVL.xIn1407 <-> Channel 8/Input
//     IO_Task Inputs/InputOutput_GVL.xIn1408 <-> Channel 9/Input
//     IO_Task Inputs/InputOutput_GVL.xIn1409 <-> Channel 10/Input
//     IO_Task Inputs/InputOutput_GVL.xIn1410 <-> Channel 11/Input
//     IO_Task Inputs/InputOutput_GVL.xIn1414 <-> Channel 15/Input
//     IO_Task Inputs/InputOutput_GVL.xIn1415 <-> Channel 16/Input
//     Monitoring_Task Inputs/InputOutput_GVL.xIn1411 <-> Channel 12/Input
//     Monitoring_Task Inputs/InputOutput_GVL.xIn1412 <-> Channel 13/Input
//     Monitoring_Task Inputs/InputOutput_GVL.xIn1413 <-> Channel 14/Input
//   Robotic/Robotic Instance <-> Main Panel (EtherCAT)/Term 1 (EK1200)/Term 5 (EL1809)
//     IO_Task Inputs/InputOutput_GVL.xIn{1500..1509} <-> Channel {1..10}/Input  (10 links)
//     Monitoring_Task Inputs/InputOutput_GVL.xIn{1510..1515} <-> Channel {11..16}/Input  (6 links)
//   Robotic/Robotic Instance <-> Main Panel (EtherCAT)/Term 1 (EK1200)/Term 6 (EL2809)
//     IO_Task Outputs/InputOutput_GVL.xOut{2000..2009} <-> Channel {1..10}/Output  (10 links)
//     Monitoring_Task Outputs/InputOutput_GVL.xOut{2010..2015} <-> Channel {11..16}/Output  (6 links)
//   Robotic/Robotic Instance <-> Main Panel (EtherCAT)/Term 1 (EK1200)/Term 7 (EL2809)
//     IO_Task Outputs/InputOutput_GVL.xOut2200 <-> Channel 1/Output
//     IO_Task Outputs/InputOutput_GVL.xOut2202 <-> Channel 3/Output
//     IO_Task Outputs/InputOutput_GVL.xOut2203 <-> Channel 4/Output
//     IO_Task Outputs/InputOutput_GVL.xOut2204 <-> Channel 5/Output
//     IO_Task Outputs/InputOutput_GVL.xOut2205 <-> Channel 6/Output
//     IO_Task Outputs/InputOutput_GVL.xOut2207 <-> Channel 8/Output
//     IO_Task Outputs/InputOutput_GVL.xOut2208 <-> Channel 9/Output
//     IO_Task Outputs/InputOutput_GVL.xOut2209 <-> Channel 10/Output
//     IO_Task Outputs/InputOutput_GVL.xOut2210 <-> Channel 11/Output
//     IO_Task Outputs/InputOutput_GVL.xOut2215 <-> Channel 16/Output
//     Monitoring_Task Outputs/InputOutput_GVL.xOut2201 <-> Channel 2/Output
//     Monitoring_Task Outputs/InputOutput_GVL.xOut2206 <-> Channel 7/Output
//     Monitoring_Task Outputs/InputOutput_GVL.xOut2211 <-> Channel 12/Output
//     Monitoring_Task Outputs/InputOutput_GVL.xOut2212 <-> Channel 13/Output
//     Monitoring_Task Outputs/InputOutput_GVL.xOut2213 <-> Channel 14/Output
//     Monitoring_Task Outputs/InputOutput_GVL.xOut2214 <-> Channel 15/Output
//   Robotic/Robotic Instance <-> Main Panel (EtherCAT)/Term 1 (EK1200)/Term 8 (EL2809)
//     IO_Task Outputs/InputOutput_GVL.xOut2300 <-> Channel 1/Output
//     IO_Task Outputs/InputOutput_GVL.xOut2301 <-> Channel 2/Output
//     IO_Task Outputs/InputOutput_GVL.xOut2302 <-> Channel 3/Output
//     IO_Task Outputs/InputOutput_GVL.xOut2309 <-> Channel 10/Output
//     IO_Task Outputs/InputOutput_GVL.xOut2314 <-> Channel 15/Output
//     IO_Task Outputs/InputOutput_GVL.xOut2315 <-> Channel 16/Output
//     Monitoring_Task Outputs/InputOutput_GVL.xOut2303 <-> Channel 4/Output
//     Monitoring_Task Outputs/InputOutput_GVL.xOut2304 <-> Channel 5/Output
//     Monitoring_Task Outputs/InputOutput_GVL.xOut2305 <-> Channel 6/Output
//     Monitoring_Task Outputs/InputOutput_GVL.xOut2306 <-> Channel 7/Output
//     Monitoring_Task Outputs/InputOutput_GVL.xOut2307 <-> Channel 8/Output
//     Monitoring_Task Outputs/InputOutput_GVL.xOut2308 <-> Channel 9/Output
//     Monitoring_Task Outputs/InputOutput_GVL.xOut2310 <-> Channel 11/Output
//     Monitoring_Task Outputs/InputOutput_GVL.xOut2311 <-> Channel 12/Output
//     Monitoring_Task Outputs/InputOutput_GVL.xOut2312 <-> Channel 13/Output
//     Monitoring_Task Outputs/InputOutput_GVL.xOut2313 <-> Channel 14/Output

CONFIGURATION Robotic
    RESOURCE PLC ON TwinCAT3
        TASK Ethernet_Task(INTERVAL := T#100000us, PRIORITY := 3);
        TASK IO_Task(INTERVAL := T#2ms, PRIORITY := 1);
        TASK Main_Task(INTERVAL := T#4ms, PRIORITY := 2);
        TASK Monitoring_Task(INTERVAL := T#10ms, PRIORITY := 10);
        TASK VISU_TASK(INTERVAL := T#100000us, PRIORITY := 30);
        PROGRAM IO_Mapping WITH IO_Task : IO_Mapping;
        PROGRAM Backbone WITH Main_Task : Backbone;
        PROGRAM EM01_Robot WITH Main_Task : EM01_Robot;
        PROGRAM EM02_Placing1 WITH Main_Task : EM02_Placing1;
        PROGRAM EM03_Placing2 WITH Main_Task : EM03_Placing2;
        PROGRAM EM04_Placing3 WITH Main_Task : EM04_Placing3;
        PROGRAM EM05_Placing4 WITH Main_Task : EM05_Placing4;
        PROGRAM EM06_Picking WITH Main_Task : EM06_Picking;
        PROGRAM Module_Status WITH Monitoring_Task : Module_Status;
        PROGRAM VisuElems_Visu_Prg WITH VISU_TASK : VisuElems.Visu_Prg;
    END_RESOURCE
END_CONFIGURATION

// ---- DUTs/OEE/ShiftTime.TcDUT
TYPE ShiftTime :	
STRUCT
	Running		: TIME;
	Stopped		: TIME;
	Error		: TIME;
	sRunning	: STRING;
	sStopped	: STRING;
	sError		: STRING;
END_STRUCT
END_TYPE

// ---- DUTs/OEE/Precentage_Time.TcDUT
TYPE Precentage_Time :	
STRUCT
	Running		: REAL;
	Stopped		: REAL;
	Error		: REAL;
	Unstated	: REAL;
END_STRUCT
END_TYPE

// ---- DUTs/OEE/ShiftCounter.TcDUT
TYPE ShiftCounter :	
STRUCT
	Data1		: UINT;
	Data2		: UINT;
	Data3		: UINT;
	Data4		: UINT;
	ProductCode	: STRING(31);
END_STRUCT
END_TYPE

// ---- DUTs/OEE/sOEECounter.TcDUT
TYPE sOEECounter :	
STRUCT
	CounterRecord		: ARRAY[0..6,0..2] OF ShiftCounter;
	DateRecord			: ARRAY[0..6] OF DATE;
	HMI_Counter			: ARRAY[0..2] OF ShiftCounter;
	TimeShift			: ARRAY[1..3] OF StartShift_EndShift;				
	HMI_Date			: DATE;
	HMI_NumberLine		: UINT;
	HMI_NumberPrev		: UINT;
	CurrentShift		: UINT;
	DateCurrent			: DATE;
	TimeCurrent			: TIME_OF_DAY;
	Reset				: BOOL;
	ChangeShift			: BOOL;
	TotalCounter		: ShiftCounter;							
END_STRUCT
END_TYPE

// ---- DUTs/OEE/StartShift_EndShift.TcDUT
TYPE StartShift_EndShift :	
STRUCT
	StartShift			: TIME_OF_DAY;
	EndShift			: TIME_OF_DAY;				
END_STRUCT
END_TYPE

// ---- DUTs/OEE/sOEETime.TcDUT
TYPE sOEETime :	
STRUCT
	RecordTime			: ARRAY[0..6,0..2] OF ShiftTime;
	RecordDate			: ARRAY[0..6] OF DATE;
	HMI_Time			: ARRAY[0..2] OF ShiftTime;
	TimeShift			: ARRAY[1..3] OF StartShift_EndShift;				
	HMI_Date			: DATE;
	HMI_NumberPrev		: UINT;
	CurrentShift		: UINT;
	DateCurrent			: DATE;
	TimeCurrent			: TIME_OF_DAY;
	Reset				: BOOL;
	TotalTime			: ShiftTime;
	Precentage			: ARRAY[0..2] OF Precentage_Time;							
END_STRUCT
END_TYPE

// ---- DUTs/Robot/stCustomPattern.TcDUT
TYPE stCustomPattern :
STRUCT
	Offset_X		: ARRAY [1..24] OF INT;
	Offset_Y		: ARRAY [1..24] OF INT;
	Offset_Z		: ARRAY [1..24] OF INT;
END_STRUCT
END_TYPE

// ---- DUTs/Robot/stProductInfo.TcDUT
TYPE stProductInfo :
	STRUCT
		ProductName				: STRING;
		BarcodeReference		: STRING;
		EANVariant				: STRING;
		LinkUpSource			: STRING;
		CodeVariant				: STRING;
		ProductLength			: UINT;
		ProductWidth			: UINT;
		ProductHeight			: UINT;
		ProductPattern			: USINT;
		Stacking				: UINT;
		OffsetPattern			: stCustomPattern;
	END_STRUCT
END_TYPE

// ---- DUTs/Robot/stRobot_Input.TcDUT
TYPE stRobot_Input :
STRUCT
	StsAutoOn			: BOOL;
	StsCycleOn			: BOOL;
	StsEmergencyStop	: BOOL;
	StsMotorOn			: BOOL;
	StsMotorOff			: BOOL;
	StsExecutionError	: BOOL;
	StsSupervision		: BOOL;
	Spare1				: BOOL;
	DoneHoming			: BOOL;
	MovePicknPlaceL1	: BOOL;
	MovePicknPlaceL2	: BOOL;
	MovePicknPlaceL3	: BOOL;
	MovePicknPlaceL4	: BOOL;
	MoveReject			: BOOL;
	BusyPick			: BOOL;
	Spare4				: BOOL;
	DonePickL1			: BOOL;
	DonePickL2			: BOOL;
	DonePickL3			: BOOL;
	DonePickL4			: BOOL;
	DonePlaceL1			: BOOL;
	DonePlaceL2			: BOOL;
	DonePlaceL3			: BOOL;
	DonePlaceL4			: BOOL;
	ErrorClampOpen		: BOOL;
	ErrorTopVacuumRtc	: BOOL;
	ErrorTopVacuumAdv	: BOOL;
	ErrorTopVacuum		: BOOL;
	ErrorSideVacuum		: BOOL;
	ErrorDetectBox		: BOOL;
END_STRUCT
END_TYPE

// ---- DUTs/Robot/stRobot_Output.TcDUT
TYPE stRobot_Output :
STRUCT
	TrigMotorOn				: BOOL;
	TrigMotorOff			: BOOL;
	TrigStartProgram		: BOOL;
	TrigStartProgramAtMain	: BOOL;
	TrigStopProgram			: BOOL;
	TrigSysRestart			: BOOL;
	ResetEmergencyStop		: BOOL;
	ResetExecutionError		: BOOL;
	TrigHoming				: BOOL;
	TrigRunning				: BOOL;
	Pick					: BOOL;
	Place1					: BOOL;
	Place2					: BOOL;
	Place3					: BOOL;
	Place4					: BOOL;
	RejectBox				: BOOL;
	TestMainVacuum			: BOOL;
	TestClampOpen			: BOOL;
	TestClampClose			: BOOL;
	TestClampMid			: BOOL;
	TestSideVacuum			: BOOL;
	TestTopPneuUp			: BOOL;
	TestTopPneuDown			: BOOL;
	Spare1					: BOOL;
	BypassCheckBox			: BOOL;
	RotatePick				: BOOL;
	CheckBigBox				: BOOL;
	DoneScan1				: BOOL;
	DoneScan2				: BOOL;
	DoneScan3				: BOOL;
	DoneScan4				: BOOL;
	CheckSmallBox			: BOOL;
	GotoLine				: USINT;
	CounterL1				: USINT;
	CounterL2				: USINT;
	CounterL3				: USINT;
	CounterL4				: USINT;
	LengthL1				: unMyUINT;
	WidthL1					: unMyUINT;
	HeightL1				: unMyUINT;
	LengthL2				: unMyUINT;
	WidthL2					: unMyUINT;
	HeightL2				: unMyUINT;
	LengthL3				: unMyUINT;
	WidthL3					: unMyUINT;
	HeightL3				: unMyUINT;
	LengthL4				: unMyUINT;
	WidthL4					: unMyUINT;
	HeightL4				: unMyUINT;
	PatternL1				: USINT;
	PatternL2				: USINT;
	PatternL3				: USINT;
	PatternL4				: USINT;
	CustomX1				: unMyUINT;
	CustomY1				: unMyUINT;
	CustomX2				: unMyUINT;
	CustomY2				: unMyUINT;
	CustomX3				: unMyUINT;
	CustomY3				: unMyUINT;
	CustomX4				: unMyUINT;
	CustomY4				: unMyUINT;
	TimerClampClose			: unMyUINT;
	RotatePickInt			: USINT;
	BoxType					: USINT;
END_STRUCT
END_TYPE

// ---- DUTs/Robot/unMyINT.TcDUT
TYPE unMyINT :
UNION
	nINT	: INT;
	nSINT	: ARRAY[1..2] OF SINT;
END_UNION
END_TYPE

// ---- DUTs/Robot/unMyUINT.TcDUT
TYPE unMyUINT :
UNION
	nUINT	: UINT;
	nUSINT	: ARRAY[1..2] OF USINT;
END_UNION
END_TYPE

// ---- DUTs/stCheckShuttle.TcDUT
TYPE stCheckShuttle :
STRUCT
	AtEmpty	: BOOL;
	AtLoad	: BOOL;
END_STRUCT
END_TYPE

// ---- DUTs/stDM_Input.TcDUT
TYPE stDM_Input :
	
STRUCT
	TriggerReady			: BOOL;
	TriggerAck				: BOOL;
	Acquiring				: BOOL;
	MissedAcq				: BOOL;
	Decoding				: BOOL;
	DecodeComplete			: BOOL;
	ResultsBufferOverrun	: BOOL;
	ResultsAvailable		: BOOL;
	GeneralFault			: BOOL;
	TriggerID				: UINT;
	ResultID				: UINT;
	ResultCode				: UINT;
	ResultExtended			: UINT;
	ResultDataLength		: UINT;
	ResultData				: ARRAY [0..479] OF BYTE;
END_STRUCT

END_TYPE

// ---- DUTs/stDM_Output.TcDUT
TYPE stDM_Output :
	
STRUCT
	TriggerEnable		: BOOL;
	Trigger				: BOOL;
	BufferResultsEnable	: BOOL;
	ResultsAck			: BOOL;
	UserDataOption		: UINT;
	UserDataLength		: UINT;
	UserData			: ARRAY [0..487] OF BYTE;
END_STRUCT

END_TYPE

// ---- DUTs/stEcSlaveState.TcDUT
TYPE stEcSlaveState :
STRUCT
	ERROR		: BOOL;
	Init 		: BOOL;
	PROCESSING 	: BOOL;
	OP          : BOOL;
	
END_STRUCT
END_TYPE

// ---- DUTs/stErrorData.TcDUT
 TYPE stErrorData :
STRUCT
	Status		: UINT;
	ErrorID		: UINT;
	ErrorMsg	: STRING;
	TimeStop	: STRING;
END_STRUCT
END_TYPE

// ---- DUTs/stMachineState.TcDUT
TYPE stMachineState :
STRUCT
	Error 		: BOOL;
	CheckSafety	: BOOL;
	Aborted		: BOOL;
	Initialize	: BOOL;
	CheckToRun	: BOOL;
	Ready		: BOOL;
	Running		: BOOL;
	Stopped		: BOOL;
	ManualMode	: BOOL;
END_STRUCT
END_TYPE

// ---- DUTs/stMotor.TcDUT
TYPE stMotor :	
STRUCT
	Name				: STRING;
	TestModeActive		: BOOL;
	UseReverse			: BOOL;
	iTestForward		: BOOL;
	iTestReverse		: BOOL;
	oMoveForward		: BOOL;
	oMoveReverse		: BOOL;
	oResetError			: BOOL;
	Status_MotorRunning	: BOOL;
	Status_Error		: BOOL;
	ErrorID				: UINT;
	RunningTIME			: LTIME;
	RunningHours		: LREAL;
END_STRUCT
END_TYPE

// ---- DUTs/stPalletTrackingData.TcDUT
TYPE stPalletTrackingData :
STRUCT
	PalletID					: STRING;
	CounterProduct				: UINT;
	EANVariant					: STRING;
	CodeVariant					: STRING;
	ProductDescription			: STRING;
	PalletCreationDate			: DATE_AND_TIME;
	BarcodeProduct				: ARRAY [1..60] OF STRING;
	BarcodeProductTime			: ARRAY [1..60] OF DT;
END_STRUCT
END_TYPE

// ---- DUTs/stPneumatic1.TcDUT
TYPE stPneumatic1 : //v1.0
// UDT untuk merepresentasikan faceplate pneumatic valve 1 coil
//	Changelog:
	(* 
	v1.0 [27.12.2021] Start development UDT - Fabrilian Asali	*)	


STRUCT
	Name			: STRING;
	TestModeActive	: BOOL;
	iTest			: BOOL;
	iSensorRetract	: BOOL;
	iSensorAdvanced	: BOOL;
	oPneumatic		: BOOL;
	Trigger_Retract	: BOOL;
	Trigger_Advanced: BOOL;
	FBDone_Retract	: BOOL;
	FBDone_Advanced	: BOOL;
	ErrorRetract	: BOOL;
	ErrorAdvanced	: BOOL;
	CyclePneu		: DINT;
END_STRUCT
END_TYPE

// ---- DUTs/stPneumatic2.TcDUT
TYPE stPneumatic2 :	//v1.0
// UDT untuk merepresentasikan faceplate pneumatic valve 1 coil
//	Changelog:
	(* 
	v1.0 [27.12.2021] Start development UDT - Fabrilian Asali	*)	

STRUCT
	Name				: STRING;
	
	TestModeActive		: BOOL;
	iTestRetract		: BOOL;
	iTestAdvanced		: BOOL;
	
	iSensorRetract		: BOOL;
	iSensorAdvanced		: BOOL;
	
	oPneumaticRetract	: BOOL;
	oPneumaticAdvanced	: BOOL;
	
	Trigger_Retract		: BOOL;
	Trigger_Advanced	: BOOL;
	FB_DoneRetract		: BOOL;
	FB_DoneAdvanced		: BOOL;
	
	Error_Retract		: BOOL;
	Error_Advanced		: BOOL;
	
	CyclePneuAdv		: DINT;
	CyclePneuRtc		: DINT;
END_STRUCT
END_TYPE

// ---- DUTs/stRejectData.TcDUT
TYPE stRejectData :
STRUCT
	Status		: UINT;
	RejectID	: INT;
	RejectType	: STRING;
	Counter		: UINT;
	RejectMsg	: STRING;
	Timestamp	: STRING;
END_STRUCT
END_TYPE

// ---- DUTs/stRTC_Data.TcDUT
TYPE stRTC_Data :
STRUCT
	
	iDT_Year: INT;
	iDT_Month: INT;
	iDT_day: INT;
	iDT_Date: INT;
	iDT_Hour: INT;
	iDT_Minute: INT;
	iDT_Second: INT;
	iDT_MilliSecond: INT;
	
	strDT_Year: STRING;
	strDT_Month: STRING;
	strDT_Day: STRING;
	strDT_Date: STRING;
	strDT_Hour: STRING;
	strDT_Minute: STRING;
	strDT_Second: STRING;
	strDT_MilliSecond: STRING;
END_STRUCT
END_TYPE

// ---- DUTs/stShuttle.TcDUT
TYPE stShuttle :
STRUCT
	RequestEmptyPallet	: BOOL;
	RequestLoadPallet	: BOOL;
	FB_Request			: BOOL;
	PositionEmpty		: UINT;
	PositionLoaded		: UINT;
END_STRUCT
END_TYPE

// ---- DUTs/stDataPallet.TcDUT
TYPE stDataPallet :
STRUCT
	BarcodePallet 					: STRING; 
	BarcodePalletTime 				: DT;
END_STRUCT
END_TYPE

// ---- GVLs/Data_GVL.TcGVL
{attribute 'qualified_only'}
VAR_GLOBAL
	RTC_DATA						: stRTC_Data;
	AmsNetId_PLC					: T_AmsNetId;
	EthernetMaster 					: Tc2_System.T_AmsNetID := '';
	EtherCatMaster_D1  				: Tc2_System.T_AmsNetID := '192.168.0.119.2.1';
	stEcSlave 						: ARRAY [1..10] OF stEcSlaveState;
	
	//Init Robot
	stStateMachineRobot				: stMachineState;
	bFL_AckRobot					: BOOL;
	bFL_ResetRobot					: BOOL;
	bFL_StartRobot					: BOOL;
	bFL_StopRobot					: BOOL;
	bFL_MachineErrorRobot			: BOOL;
	bFL_AutoManuaModeRobot			: BOOL;
	StateMachineRobot_Error			: BOOL;
	StateMachineRobot_ErrorMsg		: STRING;
	StateMachineRobot_stsMachine	: STRING;
	
	//Init Picking
	stStateMachinePicking			: stMachineState;
	bFL_AckPicking					: BOOL;
	bFL_ResetPicking				: BOOL;
	bFL_StartPicking				: BOOL;
	bFL_StopPicking					: BOOL;
	bFL_MachineErrorPicking			: BOOL;
	bFL_AutoManuaModePicking		: BOOL;
	StateMachinePicking_Error		: BOOL;
	StateMachinePicking_ErrorMsg	: STRING;
	StateMachinePicking_stsMachine	: STRING;
	
	//Init Placing1
	stStateMachinePlacing1			: stMachineState;
	bFL_AckPlacing1					: BOOL;
	bFL_ResetPlacing1				: BOOL;
	bFL_StartPlacing1				: BOOL;
	bFL_StopPlacing1				: BOOL;
	bFL_MachineErrorPlacing1		: BOOL;
	bFL_AutoManuaModePlacing1		: BOOL;
	StateMachinePlacing1_Error		: BOOL;
	StateMachinePlacing1_ErrorMsg	: STRING;
	StateMachinePlacing1_stsMachine	: STRING;
	
	//Init Placing2
	stStateMachinePlacing2			: stMachineState;
	bFL_AckPlacing2					: BOOL;
	bFL_ResetPlacing2				: BOOL;
	bFL_StartPlacing2				: BOOL;
	bFL_StopPlacing2				: BOOL;
	bFL_MachineErrorPlacing2		: BOOL;
	bFL_AutoManuaModePlacing2		: BOOL;
	StateMachinePlacing2_Error		: BOOL;
	StateMachinePlacing2_ErrorMsg	: STRING;
	StateMachinePlacing2_stsMachine	: STRING;
	
	//Init Placing3
	stStateMachinePlacing3			: stMachineState;
	bFL_AckPlacing3					: BOOL;
	bFL_ResetPlacing3				: BOOL;
	bFL_StartPlacing3				: BOOL;
	bFL_StopPlacing3				: BOOL;
	bFL_MachineErrorPlacing3		: BOOL;
	bFL_AutoManuaModePlacing3		: BOOL;
	StateMachinePlacing3_Error		: BOOL;
	StateMachinePlacing3_ErrorMsg	: STRING;
	StateMachinePlacing3_stsMachine	: STRING;
	
	//Init Placing4
	stStateMachinePlacing4			: stMachineState;
	bFL_AckPlacing4					: BOOL;
	bFL_ResetPlacing4				: BOOL;
	bFL_StartPlacing4				: BOOL;
	bFL_StopPlacing4				: BOOL;
	bFL_MachineErrorPlacing4		: BOOL;
	bFL_AutoManuaModePlacing4		: BOOL;
	StateMachinePlacing4_Error		: BOOL;
	StateMachinePlacing4_ErrorMsg	: STRING;
	StateMachinePlacing4_stsMachine	: STRING;
	
	stStateMachineOutfeed			: stMachineState;
	bGetData						: ARRAY [1..4] OF BOOL;
	(*===============Request==================*)
	
	
	(*===============Feedback==================*)
	
	
	
END_VAR

VAR_GLOBAL PERSISTENT
	(**============= Timer ================*)
	Tmr_Picking		: TIME;
	Tmr_Centering	: TIME;
	Tmr_Placing1	: TIME;
	Tmr_Placing2	: TIME;
	Tmr_Placing3	: TIME;
	Tmr_Placing4	: TIME;
	
	dt_OEETime		: sOEETime;
	dt_OEEOutfeed	: sOEETime;
	dt_OEECounter	: ARRAY [1..4] OF sOEECounter;
	dt_Production	: ARRAY [1..4] OF ShiftCounter;
	UpTime			: TIME;
	UpTimeOutfeed	: TIME;
	
END_VAR

// ---- GVLs/HMI_GVL.TcGVL
{attribute 'qualified_only'}
VAR_GLOBAL
	//HMI Button Robot
	bStartButtonRobot			: BOOL;
	bStopButtonRobot			: BOOL;
	bResetButtonRobot			: BOOL;
	bTestModeEnableRobot		: BOOL;
	bAcknowledgeButtonRobot		: BOOL;
	
	//HMI Button Picking
	bStartButtonPicking			: BOOL;
	bStopButtonPicking			: BOOL;
	bResetButtonPicking			: BOOL;
	bTestModeEnablePicking		: BOOL;
	bAcknowledgeButtonPicking	: BOOL;
	bAutoStartPicking			: BOOL;
	bAutoResetPicking			: BOOL;
	bAutoAcknowledgePicking		: BOOL;
	
	//HMI Button Placing 1
	bStartButtonPlacing1		: BOOL;
	bStopButtonPlacing1			: BOOL;
	bResetButtonPlacing1		: BOOL;
	bTestModeEnablePlacing1		: BOOL;
	bAcknowledgeButtonPlacing1	: BOOL;
	
	//HMI Button Placing 2
	bStartButtonPlacing2		: BOOL;
	bStopButtonPlacing2			: BOOL;
	bResetButtonPlacing2		: BOOL;
	bTestModeEnablePlacing2		: BOOL;
	bAcknowledgeButtonPlacing2	: BOOL;
	
	//HMI Button Placing 3
	bStartButtonPlacing3		: BOOL;
	bStopButtonPlacing3			: BOOL;
	bResetButtonPlacing3		: BOOL;
	bTestModeEnablePlacing3		: BOOL;
	bAcknowledgeButtonPlacing3	: BOOL;
	
	//HMI Button Placing 4
	bStartButtonPlacing4		: BOOL;
	bStopButtonPlacing4			: BOOL;
	bResetButtonPlacing4		: BOOL;
	bTestModeEnablePlacing4		: BOOL;
	bAcknowledgeButtonPlacing4	: BOOL;
	
	//HMI Button Outfeed
	bStartButtonOutfeed			: BOOL;
	bStopButtonOutfeed			: BOOL;
	bResetButtonOutfeed			: BOOL;
	bTestModeEnableOutfeed		: BOOL;
	bAcknowledgeButtonOutfeed	: BOOL;
	
	//HMI Button Shuttle
	bStartButtonShuttle			: BOOL;
	bStopButtonShuttle			: BOOL;
	bResetButtonShuttle			: BOOL;
	bTestModeEnableShuttle		: BOOL;
	bAcknowledgeButtonShuttle	: BOOL;
	
	//HMI Button Dispenser
	bStartButtonDispenser		: BOOL;
	bStopButtonDispenser		: BOOL;
	bResetButtonDispenser		: BOOL;
	bTestModeEnableDispenser	: BOOL;
	bAcknowledgeButtonDispenser	: BOOL;
	
	//HMI Button Infeed
	bStartButtonInfeed			: BOOL;
	bStopButtonInfeed			: BOOL;
	bResetButtonInfeed			: BOOL;
	bTestModeEnableInfeed		: BOOL;
	bAcknowledgeButtonInfeed	: BOOL;
	
	bMuteBuzzer					: BOOL;
	bMachineError				: BOOL;
	sMessageError				: STRING;
	sWiringNo					: STRING;
	sCurrentJob					: STRING;
	iSeqIndex					: INT;
	xOut_HMI_Status_EcSlave 	: ARRAY [1..10] OF BOOL;
	Reset_LinkUp				: ARRAY [1..4] OF BOOL;
	
	
	(**============= Flushing ================*)
	Flush_Placing1				: BOOL;
	Flush_Placing2				: BOOL;
	Flush_Placing3				: BOOL;
	Flush_Placing4				: BOOL;
	
	(**============= Alarm Location ================*)
	AlarmRobot_Location			: ARRAY [1..20] OF BOOL;
	AlarmPicking_Location		: ARRAY [1..20] OF BOOL;
	AlarmPlacing1_Location		: ARRAY [1..20] OF BOOL;
	AlarmPlacing2_Location		: ARRAY [1..20] OF BOOL;
	AlarmPlacing3_Location		: ARRAY [1..20] OF BOOL;
	AlarmPlacing4_Location		: ARRAY [1..20] OF BOOL;
	AlarmOutfeed_Location		: ARRAY [1..100] OF BOOL;
	
	
	(**============= Current Job ================*)
	//Infeed
	CJ_Picking					: STRING;
	
	//Placing
	CJ_Placing1					: STRING;
	CJ_Placing2					: STRING;
	CJ_Placing3					: STRING;
	CJ_Placing4					: STRING;
	
	//Shuttle
	CJ_ShuttleLoad				: STRING;
	CJ_ShuttleEmpty				: STRING;
	CJ_ShuttleManagement		: STRING;
	
	//Dispenser
	CJ_Dispenser				: STRING;
	
	
	(**============= Sequence Index ================*)
	//Infeed
	SI_Picking					: INT;
	
	//Placing
	SI_Placing1					: INT;
	SI_Placing2					: INT;
	SI_Placing3					: INT;
	SI_Placing4					: INT;
	
	(**============= Test Mode Outfeed ================*)
	//Outfeed
	Test_PalletBuffer2_Fwd		: BOOL;
	Test_PalletBuffer1_Fwd		: BOOL;
	Test_PalletOutfeed1_Fwd		: BOOL;
	Test_PalletOutfeed2_Fwd		: BOOL;
	Test_PalletOutfeed3_Fwd		: BOOL;
	Test_PalletOutfeed4_Fwd		: BOOL;
	Test_PalletOutfeed5_Fwd		: BOOL;
	Test_PalletRALifter			: BOOL;
	Test_PalletRATransfer		: BOOL;
	
	//Shuttle
	Test_ShuttleDrive_Fwd		: BOOL;
	Test_ShuttleDrive_Rev		: BOOL;
	Test_ShuttleLoad_Fwd		: BOOL;
	Test_ShuttleLoad_Rev		: BOOL;
	Test_ShuttleEmpty_Fwd		: BOOL;
	
	//Infeed
	Test_BoxInfeed_Fwd			: BOOL;
	Test_BoxStopGo_Fwd			: BOOL;
	Test_BoxBuffer1_Fwd			: BOOL;
	Test_BoxBuffer2_Fwd			: BOOL;
	Test_BoxModullar1_Fwd		: BOOL;
	Test_BoxModullar2_Fwd		: BOOL;
	Test_BoxModullar3_Fwd		: BOOL;
	Test_BoxModullar4_Fwd		: BOOL;
	Test_Stopper1				: BOOL;
	Test_Stopper2				: BOOL;
	Test_Pusher_StopGo_Adv		: BOOL;
	Test_Pusher_StopGo_Rtc		: BOOL;
	Test_Pusher_Buffer1_Adv		: BOOL;
	Test_Pusher_Buffer1_Rtc		: BOOL;
	Test_Pusher_Buffer2_Adv		: BOOL;
	Test_Pusher_Buffer2_Rtc		: BOOL;
	Test_StopperModullar_Adv	: BOOL;
	Test_StopperModullar_Rtc	: BOOL;
	
END_VAR

VAR_GLOBAL PERSISTENT
	BypassWrapper				: BOOL;
	BypassWrapperExisting		: BOOL;
	BypassFGHS					: BOOL;	
	Disable_Overflow			: BOOL;
	LockModullarToRun			: BOOL;
	PickLine					: INT;
	(**============= Timer Conveyor ================*)
	//Timer
	Tmr_Picking					: UINT;
	Tmr_Centering				: UINT;
	Tmr_Placing1				: UINT;
	Tmr_Placing2				: UINT;
	Tmr_Placing3				: UINT;
	Tmr_Placing4				: UINT;
	
	(**============= Data Counter ================*)
	arCountPlace				: ARRAY [1..4] OF USINT;
	arCountReal					: ARRAY [1..4] OF USINT;
	arCountTotal				: ARRAY [1..4] OF UINT;
	arPalletIncomplete			: ARRAY [1..4] OF UINT;
	arPalletTotal				: ARRAY [1..4] OF UINT;
	
	arRecipeHMI					: ARRAY [1..4] OF stProductInfo;
	OffsetPattern1				: stCustomPattern;
	OffsetPattern2				: stCustomPattern;
	OffsetPattern3				: stCustomPattern;
	OffsetPattern4				: stCustomPattern;
	
	
	(**============= Parameter Outfeed================*)
	//Timer
	Tmr_PalletBuffer1			: UINT;
	Tmr_PalletBuffer2			: UINT;
	Tmr_PalletBuffer3			: UINT;
	Tmr_PalletOutfeed1			: UINT;
	Tmr_PalletOutfeed2			: UINT;
	Tmr_PalletOutfeed3			: UINT;
	Tmr_PalletOutfeed4			: UINT;
	Tmr_PalletOutfeed5			: UINT;
	Tmr_PalletRA				: UINT;
	TmrDelay_PalletRA			: UINT;
	Tmr_BrakeShuttle			: UINT;
	Tmr_EmptyShuttle			: UINT;
	Tmr_LoadedShuttle			: UINT;
	Tmr_Dispenser				: UINT;
	
	//Infeed
	Tmr_Infeed					: UINT;
	Tmr_Buffer1					: UINT;
	Tmr_Buffer2					: UINT;
	Tmr_StopGo					: UINT;
	Tmr_Stopper1				: UINT;
	Tmr_Stopper2				: UINT;
	Tmr_ModullarOn				: UINT;
	Tmr_ModullarOff				: UINT;
	
	(**============= Parameter Shuttle ================*)
	Shuttle_JogSpeed			: REAL;
	Shuttle_MinSpeed			: REAL;
	Shuttle_MaxSpeed			: REAL;
	Shuttle_Offset				: DINT;
	Shuttle_Speed				: REAL;
	stShuttleSequence			: ARRAY [0..4] OF stShuttle;
	LinkUp_1					: INT;
END_VAR

// ---- GVLs/InputOutput_GVL.TcGVL
{attribute 'qualified_only'}
VAR_GLOBAL
	//Barcode Reader Communication
	xIn_BarcodeReader_Picking1		AT %I* : stDM_Input;
	xOut_BarcodeReader_Picking1		AT %Q* : stDM_Output;	
	
	xIn_BarcodeReader_Picking2		AT %I* : stDM_Input;
	xOut_BarcodeReader_Picking2		AT %Q* : stDM_Output;

	xIn_BarcodeReader_Picking3		AT %I* : stDM_Input;
	xOut_BarcodeReader_Picking3		AT %Q* : stDM_Output;	
	
	xIn_BarcodeReader_Picking4		AT %I* : stDM_Input;
	xOut_BarcodeReader_Picking4		AT %Q* : stDM_Output;
	
	xIn_BarcodeReader_Picking2B		AT %I* : stDM_Input;
	xOut_BarcodeReader_Picking2B	AT %Q* : stDM_Output;
	
	xIn_BarcodeReader_Picking3B		AT %I* : stDM_Input;
	xOut_BarcodeReader_Picking3B	AT %Q* : stDM_Output;	
	
	BarcodeReader_Picking1_State	AT %I*	: UINT;
	BarcodeReader_Picking2_State	AT %I*	: UINT;
	BarcodeReader_Picking3_State	AT %I*	: UINT;
	BarcodeReader_Picking4_State	AT %I*	: UINT;
	
	BarcodeReader_Picking2B_State	AT %I*	: UINT;
	BarcodeReader_Picking3B_State	AT %I*	: UINT;
	
	//Robot Communication
	xIn_Robot						AT %I*	: stRobot_Input;
	xOut_Robot						AT %Q*	: stRobot_Output;

	xIn_ConnectionRobot				AT %I*	: ARRAY [1..64] OF USINT;
	xOut_ConnectionRobot			AT %Q*	: ARRAY [1..64] OF USINT;

	
	
	//Subscriber Input From PLC Outfeed  
	Shuttle_stsMachine				AT %I*	: STRING(31);
	Infeed_stsMachine				AT %I*	: STRING(31);
	Outfeed_stsMachine				AT %I*	: STRING(31);
	Dispenser_stsMachine			AT %I*	: STRING(31);
	Status_EcSlave					AT %I*	: ARRAY [1..10] OF BOOL;
	Digital_Input					AT %I*	: ARRAY [1..128] OF BOOL;
	Digital_Output					AT %I*	: ARRAY [1..80] OF BOOL;
	LoadPalletGoOut					AT %I*	: BOOL;
	ShuttlePosition					AT %I*	: DINT;
	FB_RequestShuttle				AT %I*	: ARRAY [0..4] OF BOOL;
	stErrorOutfeed					AT %I*	: ARRAY [1..100] OF BOOL;
	stErrorShuttle					AT %I*	: ARRAY [1..100] OF BOOL;
	stErrorDispenser				AT %I*	: ARRAY [1..100] OF BOOL;
	stErrorInfeed					AT %I*	: ARRAY [1..100] OF BOOL;
	ErrorShuttleEmpty				AT %I*	: STRING(31);
	ErrorShuttleLoad				AT %I*	: STRING(31);
	SeqIndexOutfeed					AT %I*	: ARRAY [1..10] OF INT;
	MTBF_Motor						AT %I*	: ARRAY [1..50] OF LREAL;
	MTBF_Pneumatic					AT %I*	: ARRAY [1..25] OF UINT;
	
	//Publisher Output to PLC Outfeed
	RequestEmptyPallet				AT %Q*	: ARRAY [1..4] OF BOOL;
	RequestLoadPallet				AT %Q*	: ARRAY [1..4] OF BOOL;	
	Counter							AT %Q*	: ARRAY [1..4] OF USINT;
	
	ControlButton					AT %Q*	: ARRAY [1..20] OF BOOL;
	TmrOutfeed						AT %Q*	: ARRAY [1..25] OF UINT;
	TestMode						AT %Q*	: ARRAY [1..100] OF BOOL;
	Shuttle_Speed					AT %Q*	: ARRAY [1..4] OF REAL;
	stShuttleSequence				AT %Q*	: ARRAY [0..4] OF stShuttle;
	Shuttle_Offset					AT %Q*	: DINT;
	Error_Safety					AT %Q*	: BOOL;
	PickingBusy						AT %Q*	: BOOL;
	

	//Main Panel (P1)
	//Digital Input 16 Point EL1809
	xIn1000				AT 		%I*			: BOOL;		// Push Button Run at Main Panel
	xIn1001				AT 		%I*			: BOOL;		// Push Button Stop at Main Panel
	xIn1002				AT 		%I*			: BOOL;		// Push Button Alarm Reset at Main Panel
	xIn1003				AT 		%I*			: BOOL;		// Push Button Acknowledge at Main Panel
	xIn1004				AT 		%I*			: BOOL;		// Emergency Stop at Infeed Panel
	xIn1005				AT 		%I*			: BOOL;		// 
	xIn1006				AT 		%I*			: BOOL;		// 
	xIn1007				AT 		%I*			: BOOL;		// 
	xIn1008				AT 		%I*			: BOOL;		// 
	xIn1009				AT 		%I*			: BOOL;		// 
	xIn1010				AT 		%I*			: BOOL;		// 
	xIn1011				AT 		%I*			: BOOL;		// 
	xIn1012				AT 		%I*			: BOOL;		// 
	xIn1013				AT 		%I*			: BOOL;		// 
	xIn1014				AT 		%I*			: BOOL;		// 
	xIn1015				AT 		%I*			: BOOL;		// Pressure Switch for Main Panel

	//Digital Input 16 Point EL1809
	xIn1200				AT 		%I*			: BOOL;		// Feedback Box Picking roller Conveyor is Running
	xIn1201				AT 		%I*			: BOOL;		// 
	xIn1202				AT 		%I*			: BOOL;		// Feedback Box Placing at Pallet Roller Conveyor 1 is Running
	xIn1203				AT 		%I*			: BOOL;		// Feedback Box Placing at Pallet Roller Conveyor 2 is Running
	xIn1204				AT 		%I*			: BOOL;		// Feedback Box Placing at Pallet Roller Conveyor 3 is Running
	xIn1205				AT 		%I*			: BOOL;		// Feedback Box Placing at Pallet Roller Conveyor 4  isRunning
	xIn1206				AT 		%I*			: BOOL;		// 
	xIn1207				AT 		%I*			: BOOL;		// 
	xIn1208				AT 		%I*			: BOOL;		// 
	xIn1209				AT 		%I*			: BOOL;		// 
	xIn1210				AT 		%I*			: BOOL;		// 
	xIn1211				AT 		%I*			: BOOL;		// RSW Pneumatic Box Centering When Rtc
	xIn1212				AT 		%I*			: BOOL;		// RSW Pneumatic Gap Maker When Adv
	xIn1213				AT 		%I*			: BOOL;		// RSW Pneumatic Gap Maker When Rtc
	xIn1214				AT 		%I*			: BOOL;		// RSW Pneumatic Stopper  Transfer When Rtc
	xIn1215				AT 		%I*			: BOOL;		// 
	//Digital Input 16 Point EL1809
	xIn1400				AT 		%I*			: BOOL;		// PSR 4 to Detect Box at Picking Conv.  (GTE6-P4212)
	xIn1401				AT 		%I*			: BOOL;		// PSR to Detect Box at Barcoder Reading 2 Conv (GL6-P4212) (Not Used)
	xIn1402				AT 		%I*			: BOOL;		// PSR to Detect Box at Barcoder Reading 3 Conv (GL6-P4212) (Not Used)
	xIn1403				AT 		%I*			: BOOL;		// PSR to Detect Box at Barcoder Reading 4 Conv (GL6-P4212) (Not Used)
	xIn1404				AT 		%I*			: BOOL;		// PSR to Detect Centering Box. (GL6-P4212) (Not Used)
	xIn1405				AT 		%I*			: BOOL;		// PSR 1 to Detect Box at Picking Conv.  (GTE6-P4212)
	xIn1406				AT 		%I*			: BOOL;		// PSR 2 to Detect Box at Picking Conv. (GTE6-P4212)
	xIn1407				AT 		%I*			: BOOL;		// PSR 3 to Detect Box at Picking Conv.  (GTE6-P4212)
	xIn1408				AT 		%I*			: BOOL;		// PSR Front to Detect for Empty Transfer Infeed Roller. (GL6-P4212)
	xIn1409				AT 		%I*			: BOOL;		// PSR Middle to Detect for Empty Transfer Infeed Roller. (GL6-P4212)
	xIn1410				AT 		%I*			: BOOL;		// PSR Back to Detect for Empty Transfer Infeed Roller. (GL6-P4212)
	xIn1411				AT 		%I*			: BOOL;		// 
	xIn1412				AT 		%I*			: BOOL;		// 
	xIn1413				AT 		%I*			: BOOL;		// 
	xIn1414				AT 		%I*			: BOOL;		// Request Release Solenoid Door Robot
	xIn1415				AT 		%I*			: BOOL;		// Feedback Relay Solenoid Door Robot
	//Digital Input 16 Point EL1809
	xIn1500				AT 		%I*			: BOOL;		// PSR Back at Placing Conv 1 (GL6-P4212)
	xIn1501				AT 		%I*			: BOOL;		// PSR Middle at Placing Conv 1 (GL6-P4212)
	xIn1502				AT 		%I*			: BOOL;		// PSR Front at Placing Conv 1 (GL6-P4212)
	xIn1503				AT 		%I*			: BOOL;		// PSR Back at Placing Conv 2 (GL6-P4212)
	xIn1504				AT 		%I*			: BOOL;		// PSR Front at Placing Conv 2 (GL6-P4212)
	xIn1505				AT 		%I*			: BOOL;		// PSR Back at Placing Conv 3 (GL6-P4212)
	xIn1506				AT 		%I*			: BOOL;		// PSR Front at Placing Conv 3 (GL6-P4212)
	xIn1507				AT 		%I*			: BOOL;		// PSR Back at Placing Conv 4 (GL6-P4212)
	xIn1508				AT 		%I*			: BOOL;		// PSR Middle at Placing Conv 4 (GL6-P4212)
	xIn1509				AT 		%I*			: BOOL;		// PSR Front at Placing Conv 4 (GL6-P4212)
	xIn1510				AT 		%I*			: BOOL;		// 
	xIn1511				AT 		%I*			: BOOL;		// 
	xIn1512				AT 		%I*			: BOOL;		// 
	xIn1513				AT 		%I*			: BOOL;		// 
	xIn1514				AT 		%I*			: BOOL;		// 
	xIn1515				AT 		%I*			: BOOL;		// 
	
	
	//Main Panel (P1)
	//Digital Output 16 Point EL2809
	xOut2000			AT 		%Q*			: BOOL;		// Indicator Machine Running at Main Panel
	xOut2001			AT 		%Q*			: BOOL;		// Indicator Machine Error at Main Panel
	xOut2002			AT 		%Q*			: BOOL;		// Indicator Tower Lamp Red
	xOut2003			AT 		%Q*			: BOOL;		// Indicator Tower Lamp Yellow
	xOut2004			AT 		%Q*			: BOOL;		// Indicator Tower lamp Green
	xOut2005			AT 		%Q*			: BOOL;		// Indicator Tower lamp Blue
	xOut2006			AT 		%Q*			: BOOL;		// Indicator Buzzer
	xOut2007			AT 		%Q*			: BOOL;		// Indicator Acknowledge at Main Panel
	xOut2008			AT 		%Q*			: BOOL;		// Indicator Auto Mode Main Panel
	xOut2009			AT 		%Q*			: BOOL;		// Indicator Manual Mode Main Panel
	xOut2010			AT 		%Q*			: BOOL;		// 
	xOut2011			AT 		%Q*			: BOOL;		// 
	xOut2012			AT 		%Q*			: BOOL;		// 
	xOut2013			AT 		%Q*			: BOOL;		// 
	xOut2014			AT 		%Q*			: BOOL;		// 
	xOut2015			AT 		%Q*			: BOOL;		// 
	//Digital Output 16 Point EL2809
	xOut2200			AT 		%Q*			: BOOL;		// Move Forward for Picking Roller Conveyor
	xOut2201			AT 		%Q*			: BOOL;		// 
	xOut2202			AT 		%Q*			: BOOL;		// Move Forward for Placing At Pallet Roller Conveyor  1
	xOut2203			AT 		%Q*			: BOOL;		// Move Forward for Placing At Pallet Roller Conveyor  2
	xOut2204			AT 		%Q*			: BOOL;		// Move Forward for Placing At Pallet Roller Conveyor  3
	xOut2205			AT 		%Q*			: BOOL;		// Move Forward for Placing At Pallet Roller Conveyor  4
	xOut2206			AT 		%Q*			: BOOL;		// 
	xOut2207			AT 		%Q*			: BOOL;		// Move Reverse for Placing At Pallet Roller Conveyor  1
	xOut2208			AT 		%Q*			: BOOL;		// Move Reverse for Placing At Pallet Roller Conveyor  2
	xOut2209			AT 		%Q*			: BOOL;		// Move Reverse for Placing At Pallet Roller Conveyor  3
	xOut2210			AT 		%Q*			: BOOL;		// Move Reverse for Placing At Pallet Roller Conveyor  4
	xOut2211			AT 		%Q*			: BOOL;		// 
	xOut2212			AT 		%Q*			: BOOL;		// 
	xOut2213			AT 		%Q*			: BOOL;		// 
	xOut2214			AT 		%Q*			: BOOL;		// 
	xOut2215			AT 		%Q*			: BOOL;		// Reset Error for All Inverter at P1, Relay
	//Digital Output 16 Point EL2809
	xOut2300			AT 		%Q*			: BOOL;		// Pneumatic Box Centering
	xOut2301			AT 		%Q*			: BOOL;		// Pneumatic Gap Maker Box Adv
	xOut2302			AT 		%Q*			: BOOL;		// Pneumatic Gap Maker Box Rtc
	xOut2303			AT 		%Q*			: BOOL;		// 
	xOut2304			AT 		%Q*			: BOOL;		// 
	xOut2305			AT 		%Q*			: BOOL;		// 
	xOut2306			AT 		%Q*			: BOOL;		// 
	xOut2307			AT 		%Q*			: BOOL;		// 
	xOut2308			AT 		%Q*			: BOOL;		// 
	xOut2309			AT 		%Q*			: BOOL;		// Pneumatic Stopper Transfer
	xOut2310			AT 		%Q*			: BOOL;		// 
	xOut2311			AT 		%Q*			: BOOL;		// 
	xOut2312			AT 		%Q*			: BOOL;		// 
	xOut2313			AT 		%Q*			: BOOL;		// 
	xOut2314			AT 		%Q*			: BOOL;		// Status Solenoid Door Robot
	xOut2315			AT 		%Q*			: BOOL;		// Release Solenoid Door Robot
	
END_VAR

// ---- GVLs/Status_GVL.TcGVL
{attribute 'qualified_only'}
VAR_GLOBAL
	bFl_RunButton_Robotic	: BOOL;
	bFl_StopButton_Robotic	: BOOL;
	bFl_ResetButton_Robotic	: BOOL;
	bFl_Acknowledge_Robotic	: BOOL;
	bFl_Manual_Robotic		: BOOL;
	bFl_EStop_Robotic		: BOOL;
	bFl_ReqReleaseDoor		: BOOL;
	bFl_StsDoorReleased		: BOOL;
	
	
	//Error
	stErrorRobot			: ARRAY [1..100] OF BOOL;
	stErrorPicking			: ARRAY [1..100] OF BOOL;
	stErrorPlacing1			: ARRAY [1..100] OF BOOL;
	stErrorPlacing2			: ARRAY [1..100] OF BOOL;
	stErrorPlacing3			: ARRAY [1..100] OF BOOL;
	stErrorPlacing4			: ARRAY [1..100] OF BOOL;
	arAlarmHistory			: ARRAY [0..100] OF stErrorData;
	arAlarmActive			: ARRAY [0..100] OF stErrorData;
	arRejectMsg				: ARRAY [1..20] OF stRejectData;
	Module_Error			: ARRAY [1..10] OF BOOL;
	WarningAcc				: ARRAY [1..4] OF BOOL;
	
	bTrig_LED_MachineRunning_Robotic	: BOOL;
	bTrig_LED_MachineError_Robotic		: BOOL;
	bTrig_TowerLamp_Red_Robotic			: BOOL;
	bTrig_TowerLamp_Yellow_Robotic		: BOOL;
	bTrig_TowerLamp_Green_Robotic		: BOOL;
	bTrig_TowerLamp_Blue_Robotic		: BOOL;
	bTrig_Buzzer_Robotic				: BOOL;
	bTrig_LED_Acknowledge_Robotic		: BOOL;
	bTrig_LED_Auto_Robotic				: BOOL;
	bTrig_LED_Manual_Robotic			: BOOL;
	bTrig_LED_SafetyDoor_Robotic		: BOOL;
	
	
	(*===============Auto Flsuhing==================*)
	
	AutoFlush_Placing1					: BOOL;
	AutoFlush_Placing2					: BOOL;
	AutoFlush_Placing3					: BOOL;
	AutoFlush_Placing4					: BOOL;
	PalletOut_1							: BOOL;
	PalletOut_2							: BOOL;
	PalletOut_3							: BOOL;
	PalletOut_4							: BOOL;
	
	(*===============Safety==================*)
	bAirPressure_Robotic				: BOOL;
	bSafety_DoorRobotic					: BOOL;
	bRelease_DoorRobotic				: BOOL;
	
	
	(*=============== Data ==================*)
	BarcodeResult						: STRING;
	BarcodePlace						: INT;
	Edit								: ARRAY [1..4] OF BOOL;
	Upload								: ARRAY [1..4] OF BOOL;
	Download							: ARRAY [1..4] OF BOOL;
	Save								: ARRAY [1..4] OF BOOL;
	Cancel								: ARRAY [1..4] OF BOOL;
	StsEdit								: ARRAY [1..4] OF BOOL;
	
	QtyCyclePerLayer					: ARRAY [1..4] OF UINT;
	CurrentLayer						: ARRAY [1..4] OF UINT;
	CycleAtLayer						: ARRAY [1..4] OF UINT;
	
	
	(*=============== Status ==================*)
	
	RequestEmptyPallet					: ARRAY [1..4] OF BOOL;
	RequestLoadPallet					: ARRAY [1..4] OF BOOL;
	FB_RequestShuttle					: ARRAY [1..4] OF BOOL;
	PlacingReady						: ARRAY [1..4] OF BOOL;
	RejectReady							: BOOL;
	RejectFull							: BOOL;
	ModullarInfeedBusy					: BOOL;
	
	ErrorCollectBarcode					: ARRAY [1..4] OF BOOL;
	ErrorMsgCollectBarcode				: ARRAY [1..4] OF STRING;
	stCheckShuttlePos					: ARRAY [0..4] OF stCheckShuttle;
	 
	
	
	(*===============Feedback Motor==================*)
	//Infeed
	bFdbk_Picking				: BOOL;
	bFdbk_Placing1				: BOOL;
	bFdbk_Placing2				: BOOL;
	bFdbk_Placing3				: BOOL;
	bFdbk_Placing4				: BOOL;
	
	(*===============Reedswitch==================*)
	bRsw_Centering_Rtc			: BOOL;
	bRsw_Centering_Adv			: BOOL;
	bRsw_GapMaker_Rtc			: BOOL;
	bRsw_GapMaker_Adv			: BOOL;
	bRsw_StopperTransfer_Rtc	: BOOL;
	bRsw_StopperTransfer_Adv	: BOOL;
	
	(*===============Photosensor==================*)
	//Infeed
	bPsr_Picking1				: BOOL;
	bPsr_Picking2				: BOOL;
	bPsr_Picking3				: BOOL;
	bPsr_Picking4				: BOOL;
	bPsr_Barcode1				: BOOL;
	bPsr_Barcode2				: BOOL;
	bPsr_Barcode3				: BOOL;
	bPsr_Barcode4				: BOOL;
	bPsr_Centering				: BOOL;
	bPsr_TransferInfeed_Front	: BOOL;
	bPsr_TransferInfeed_Mid		: BOOL;
	bPsr_TransferInfeed_Back	: BOOL;
	
	//Placing
	bPsr_Placing1_Back			: BOOL;
	bPsr_Placing1_Mid			: BOOL;
	bPsr_Placing1_Front			: BOOL;
	bPsr_Placing2_Back			: BOOL;
	bPsr_Placing2_Front			: BOOL;
	bPsr_Placing3_Back			: BOOL;
	bPsr_Placing3_Front			: BOOL;
	bPsr_Placing4_Back			: BOOL;
	bPsr_Placing4_Mid			: BOOL;
	bPsr_Placing4_Front			: BOOL;
	
	
	strTimeEvent				: STRING;

END_VAR

VAR_GLOBAL PERSISTENT
	(*===============stMotor==================*)
	//Infeed
	stMotor_Picking						: stMotor;
	stMotor_Placing1					: stMotor;
	stMotor_Placing2					: stMotor;
	stMotor_Placing3					: stMotor;
	stMotor_Placing4					: stMotor;	

	(*===============Pneumatic==================*)
	stPneu_Centering					: stPneumatic1;
	stPneu_GapMaker						: stPneumatic2; 
	stPneu_StopperTransfer				: stPneumatic1;	

	(*===============Data Recipe==================*)
	RecipeLine							: ARRAY [1..4] OF stProductInfo;
	arProductList						: ARRAY [1..40] OF stProductInfo;
	RecipeNumber						: ARRAY [1..4] OF USINT;
	OffsetPattern1						: ARRAY [1..40] OF stCustomPattern;
	OffsetPattern2						: ARRAY [1..40] OF stCustomPattern;
	OffsetPattern3						: ARRAY [1..40] OF stCustomPattern;
	OffsetPattern4						: ARRAY [1..40] OF stCustomPattern;
	
	
	(*===============FGHS Var==================*)
	//To FGHS
	//==> Read Only
	arPallet_LinkUp						: ARRAY [1..4] OF STRING; // Source Link Up
	arCurrent_EAN						: ARRAY [1..4] OF STRING; // Currently used EAN
	arCurrent_CodeVariant				: ARRAY [1..4] OF STRING; // Currently used Code Variant
	arPalletID							: ARRAY [1..4] OF STRING; // Generated Pallet ID
	arBarcodePallet 					: ARRAY [1..4,1..60] OF STRING; // Array of Barcode Product at Pallet
	arBarcodePalletTime 				: ARRAY [1..4,1..60] OF DT; // Array of Placing Time Product at Pallet
	arCounterProduct					: ARRAY [1..4] OF BYTE; // Counter Product at Pallet
	arRejectList						: ARRAY [1..3] OF BOOL; // Status Reject : 1. Reject Bad Read, 2. No Match Barcode to Reference, 3. Placing Not Ready
	arAlarmList							: ARRAY [1..300] OF BOOL; // Active Alarm
	//Time
	Time_PLC							: STRING(31);
	
	//==> Full Access
	arAccFlushingPallet					: ARRAY [1..4] OF BYTE; //Status Pallet : 0. Procees Palletizing, 1. Request Pallet to Flushing, 2. Acc Flushing  
	arPlanned_EAN						: ARRAY [1..4] OF STRING; // Planned EAN for Brand Change
	arPlanned_CodeVariant				: ARRAY [1..4] OF STRING; // Planned Code Variant for Brand Change
	
	//Internal
	arPalletStackingDone				: ARRAY [1..4] OF BOOL; //Pallet Request to Flush
	arPalletizingBuffer					: ARRAY [1..4] OF stPalletTrackingData; 
	arDataPallet1						: ARRAY [1..60] OF stDataPallet;
	arDataPallet2						: ARRAY [1..60] OF stDataPallet;
	arDataPallet3						: ARRAY [1..60] OF stDataPallet;
	arDataPallet4						: ARRAY [1..60] OF stDataPallet;
END_VAR

// ---- POUs/S00_System_Utilities/IO_Mapping.TcPOU
PROGRAM IO_Mapping
VAR
	BLINK_500msOn_500MsOff	: Blink;
END_VAR

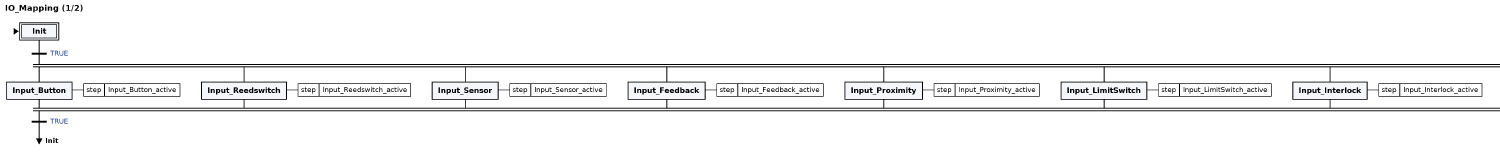
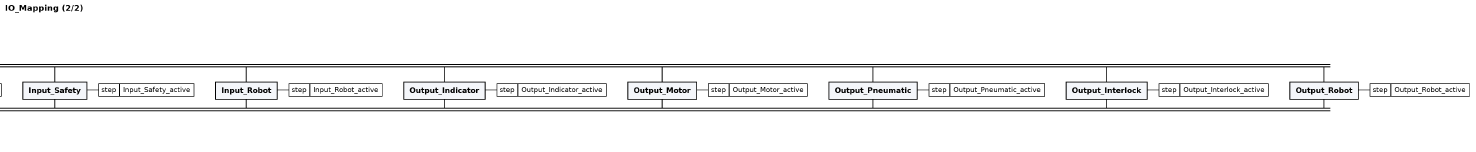
INITIAL_STEP Init:
END_STEP
TRANSITION FROM Init TO (Input_Button, Input_Reedswitch, Input_Sensor, Input_Feedback, Input_Proximity, Input_LimitSwitch, Input_Interlock, Input_Safety, Input_Robot, Output_Indicator, Output_Motor, Output_Pneumatic, Output_Interlock, Output_Robot)
    := TRUE;
END_TRANSITION
STEP Input_Button:
    Input_Button_active(N);  // step action
END_STEP
STEP Input_Reedswitch:
    Input_Reedswitch_active(N);  // step action
END_STEP
STEP Input_Sensor:
    Input_Sensor_active(N);  // step action
END_STEP
STEP Input_Feedback:
    Input_Feedback_active(N);  // step action
END_STEP
STEP Input_Proximity:
    Input_Proximity_active(N);  // step action
END_STEP
STEP Input_LimitSwitch:
    Input_LimitSwitch_active(N);  // step action
END_STEP
STEP Input_Interlock:
    Input_Interlock_active(N);  // step action
END_STEP
STEP Input_Safety:
    Input_Safety_active(N);  // step action
END_STEP
STEP Input_Robot:
    Input_Robot_active(N);  // step action
END_STEP
STEP Output_Indicator:
    Output_Indicator_active(N);  // step action
END_STEP
STEP Output_Motor:
    Output_Motor_active(N);  // step action
END_STEP
STEP Output_Pneumatic:
    Output_Pneumatic_active(N);  // step action
END_STEP
STEP Output_Interlock:
    Output_Interlock_active(N);  // step action
END_STEP
STEP Output_Robot:
    Output_Robot_active(N);  // step action
END_STEP
TRANSITION FROM (Input_Button, Input_Reedswitch, Input_Sensor, Input_Feedback, Input_Proximity, Input_LimitSwitch, Input_Interlock, Input_Safety, Input_Robot, Output_Indicator, Output_Motor, Output_Pneumatic, Output_Interlock, Output_Robot) TO Init
    := TRUE;
END_TRANSITION

ACTION Input_Button_active:
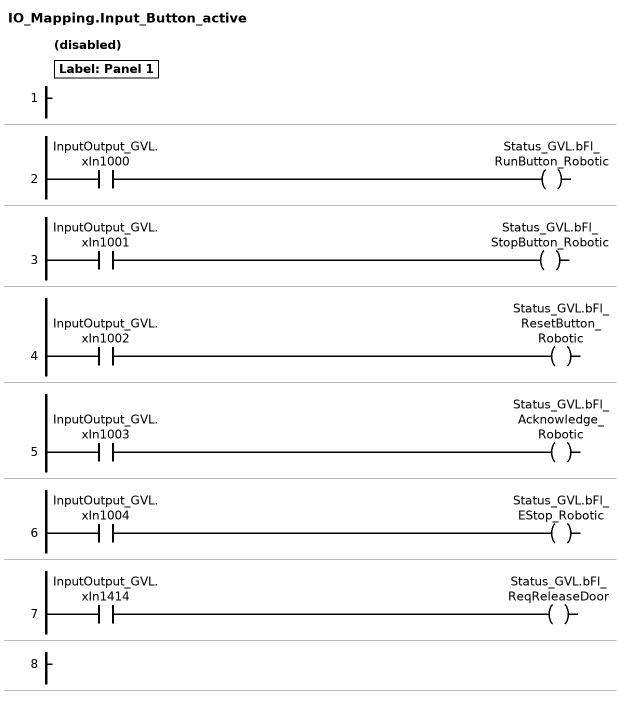
// NETWORK 1 (disabled)
// label: Label: Panel 1

// NETWORK 2
Status_GVL.bFl_RunButton_Robotic := InputOutput_GVL.xIn1000;

// NETWORK 3
Status_GVL.bFl_StopButton_Robotic := InputOutput_GVL.xIn1001;

// NETWORK 4
Status_GVL.bFl_ResetButton_Robotic := InputOutput_GVL.xIn1002;

// NETWORK 5
Status_GVL.bFl_Acknowledge_Robotic := InputOutput_GVL.xIn1003;

// NETWORK 6
Status_GVL.bFl_EStop_Robotic := InputOutput_GVL.xIn1004;

// NETWORK 7
Status_GVL.bFl_ReqReleaseDoor := InputOutput_GVL.xIn1414;

// NETWORK 8
END_ACTION

ACTION Input_Feedback_active:
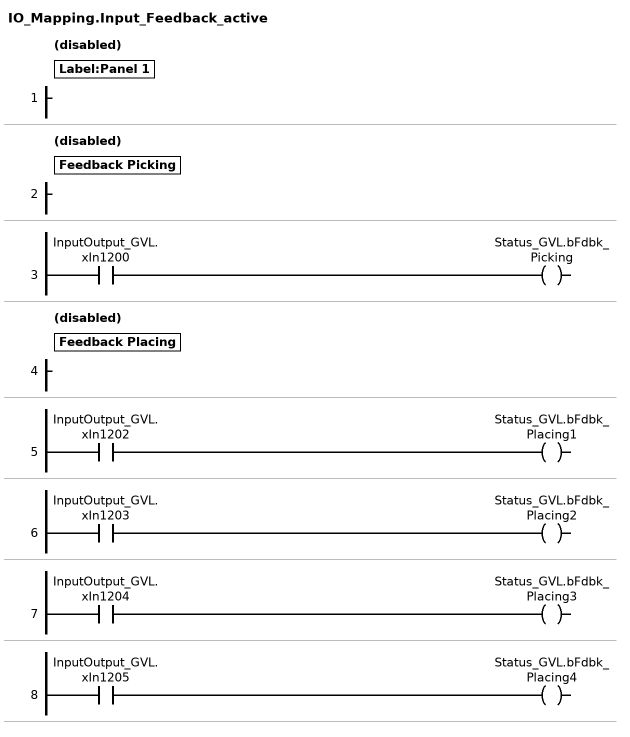
// NETWORK 1 (disabled)
// label: Label:Panel 1

// NETWORK 2 (disabled)
// label: Feedback Picking

// NETWORK 3
Status_GVL.bFdbk_Picking := InputOutput_GVL.xIn1200;

// NETWORK 4 (disabled)
// label: Feedback Placing

// NETWORK 5
Status_GVL.bFdbk_Placing1 := InputOutput_GVL.xIn1202;

// NETWORK 6
Status_GVL.bFdbk_Placing2 := InputOutput_GVL.xIn1203;

// NETWORK 7
Status_GVL.bFdbk_Placing3 := InputOutput_GVL.xIn1204;

// NETWORK 8
Status_GVL.bFdbk_Placing4 := InputOutput_GVL.xIn1205;
END_ACTION

ACTION Input_Interlock_active:
// NETWORK 1
END_ACTION

ACTION Input_LimitSwitch_active:
// NETWORK 1
END_ACTION

ACTION Input_Proximity_active:
// NETWORK 1 (disabled)
// label: Proximity

// NETWORK 2
END_ACTION

ACTION Input_Reedswitch_active:
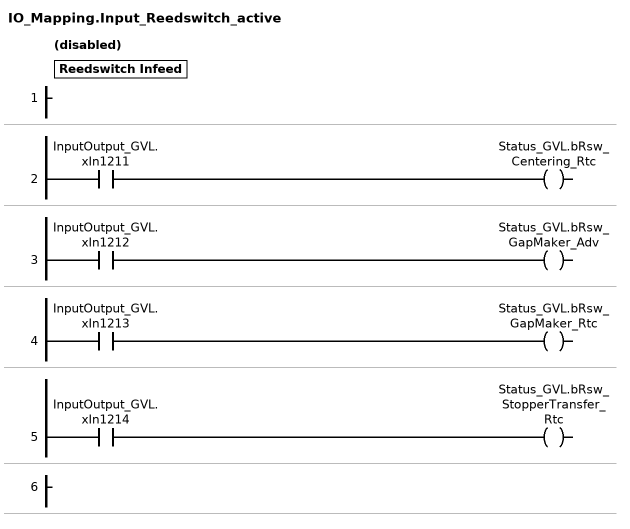
// NETWORK 1 (disabled)
// label: Reedswitch Infeed

// NETWORK 2
Status_GVL.bRsw_Centering_Rtc := InputOutput_GVL.xIn1211;

// NETWORK 3
Status_GVL.bRsw_GapMaker_Adv := InputOutput_GVL.xIn1212;

// NETWORK 4
Status_GVL.bRsw_GapMaker_Rtc := InputOutput_GVL.xIn1213;

// NETWORK 5
Status_GVL.bRsw_StopperTransfer_Rtc := InputOutput_GVL.xIn1214;

// NETWORK 6
END_ACTION

ACTION Input_Robot_active:
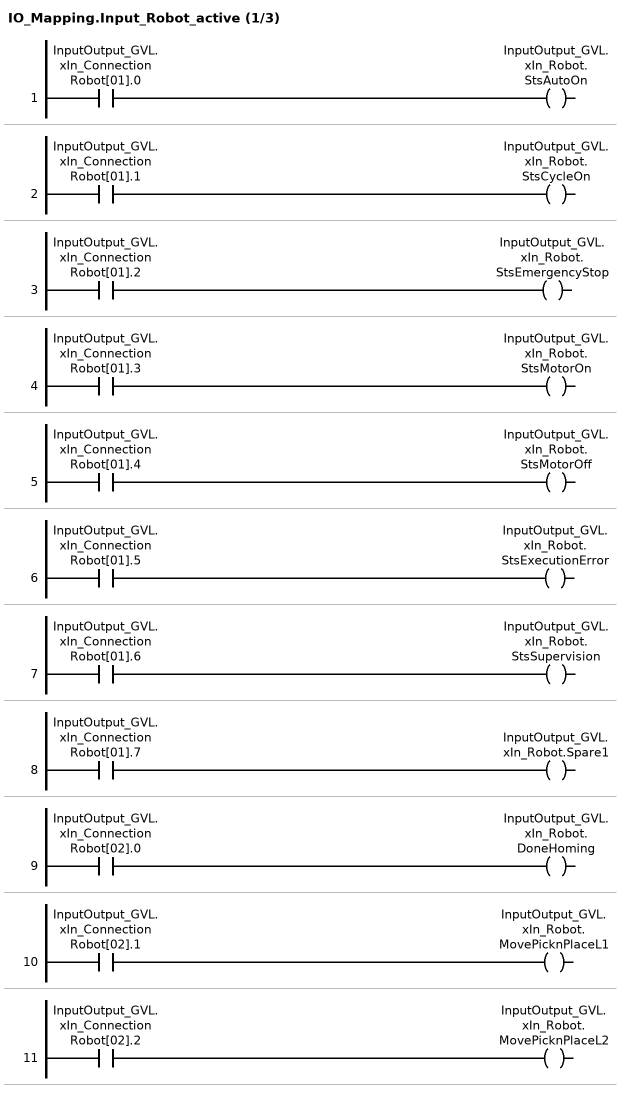
// NETWORK 1
InputOutput_GVL.xIn_Robot.StsAutoOn := InputOutput_GVL.xIn_ConnectionRobot[01].0;

// NETWORK 2
InputOutput_GVL.xIn_Robot.StsCycleOn := InputOutput_GVL.xIn_ConnectionRobot[01].1;

// NETWORK 3
InputOutput_GVL.xIn_Robot.StsEmergencyStop := InputOutput_GVL.xIn_ConnectionRobot[01].2;

// NETWORK 4
InputOutput_GVL.xIn_Robot.StsMotorOn := InputOutput_GVL.xIn_ConnectionRobot[01].3;

// NETWORK 5
InputOutput_GVL.xIn_Robot.StsMotorOff := InputOutput_GVL.xIn_ConnectionRobot[01].4;

// NETWORK 6
InputOutput_GVL.xIn_Robot.StsExecutionError := InputOutput_GVL.xIn_ConnectionRobot[01].5;

// NETWORK 7
InputOutput_GVL.xIn_Robot.StsSupervision := InputOutput_GVL.xIn_ConnectionRobot[01].6;

// NETWORK 8
InputOutput_GVL.xIn_Robot.Spare1 := InputOutput_GVL.xIn_ConnectionRobot[01].7;

// NETWORK 9
InputOutput_GVL.xIn_Robot.DoneHoming := InputOutput_GVL.xIn_ConnectionRobot[02].0;

// NETWORK 10
InputOutput_GVL.xIn_Robot.MovePicknPlaceL1 := InputOutput_GVL.xIn_ConnectionRobot[02].1;

// NETWORK 11
InputOutput_GVL.xIn_Robot.MovePicknPlaceL2 := InputOutput_GVL.xIn_ConnectionRobot[02].2;

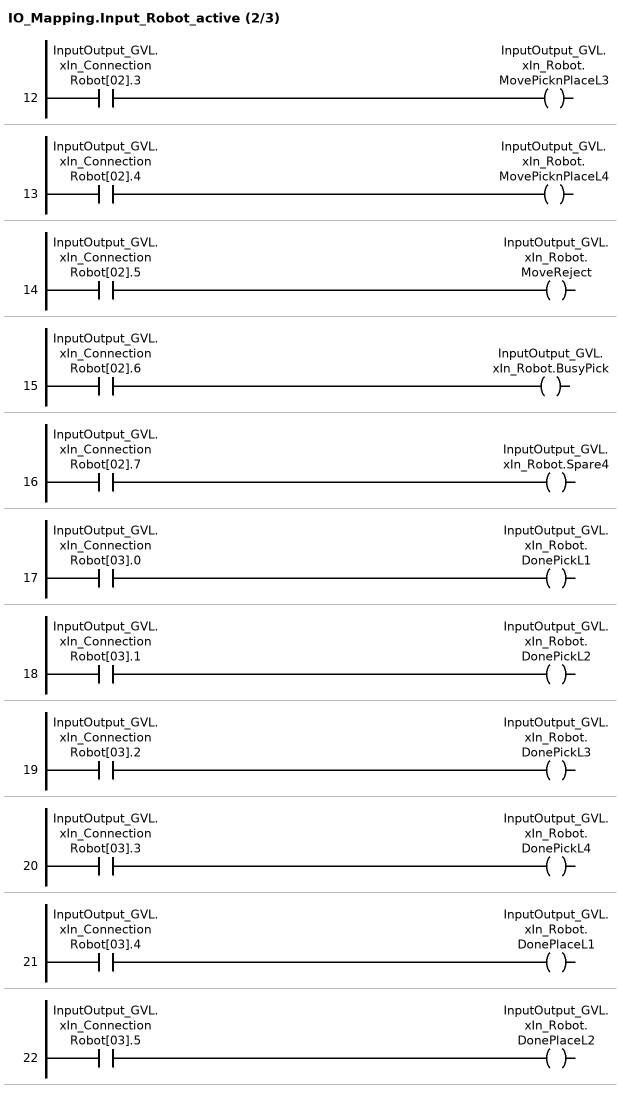
// NETWORK 12
InputOutput_GVL.xIn_Robot.MovePicknPlaceL3 := InputOutput_GVL.xIn_ConnectionRobot[02].3;

// NETWORK 13
InputOutput_GVL.xIn_Robot.MovePicknPlaceL4 := InputOutput_GVL.xIn_ConnectionRobot[02].4;

// NETWORK 14
InputOutput_GVL.xIn_Robot.MoveReject := InputOutput_GVL.xIn_ConnectionRobot[02].5;

// NETWORK 15
InputOutput_GVL.xIn_Robot.BusyPick := InputOutput_GVL.xIn_ConnectionRobot[02].6;

// NETWORK 16
InputOutput_GVL.xIn_Robot.Spare4 := InputOutput_GVL.xIn_ConnectionRobot[02].7;

// NETWORK 17
InputOutput_GVL.xIn_Robot.DonePickL1 := InputOutput_GVL.xIn_ConnectionRobot[03].0;

// NETWORK 18
InputOutput_GVL.xIn_Robot.DonePickL2 := InputOutput_GVL.xIn_ConnectionRobot[03].1;

// NETWORK 19
InputOutput_GVL.xIn_Robot.DonePickL3 := InputOutput_GVL.xIn_ConnectionRobot[03].2;

// NETWORK 20
InputOutput_GVL.xIn_Robot.DonePickL4 := InputOutput_GVL.xIn_ConnectionRobot[03].3;

// NETWORK 21
InputOutput_GVL.xIn_Robot.DonePlaceL1 := InputOutput_GVL.xIn_ConnectionRobot[03].4;

// NETWORK 22
InputOutput_GVL.xIn_Robot.DonePlaceL2 := InputOutput_GVL.xIn_ConnectionRobot[03].5;

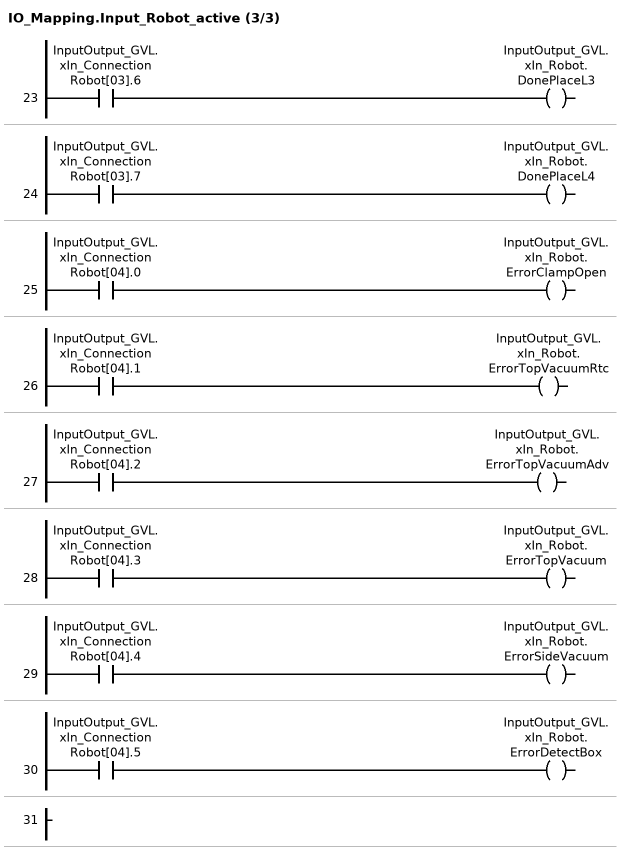
// NETWORK 23
InputOutput_GVL.xIn_Robot.DonePlaceL3 := InputOutput_GVL.xIn_ConnectionRobot[03].6;

// NETWORK 24
InputOutput_GVL.xIn_Robot.DonePlaceL4 := InputOutput_GVL.xIn_ConnectionRobot[03].7;

// NETWORK 25
InputOutput_GVL.xIn_Robot.ErrorClampOpen := InputOutput_GVL.xIn_ConnectionRobot[04].0;

// NETWORK 26
InputOutput_GVL.xIn_Robot.ErrorTopVacuumRtc := InputOutput_GVL.xIn_ConnectionRobot[04].1;

// NETWORK 27
InputOutput_GVL.xIn_Robot.ErrorTopVacuumAdv := InputOutput_GVL.xIn_ConnectionRobot[04].2;

// NETWORK 28
InputOutput_GVL.xIn_Robot.ErrorTopVacuum := InputOutput_GVL.xIn_ConnectionRobot[04].3;

// NETWORK 29
InputOutput_GVL.xIn_Robot.ErrorSideVacuum := InputOutput_GVL.xIn_ConnectionRobot[04].4;

// NETWORK 30
InputOutput_GVL.xIn_Robot.ErrorDetectBox := InputOutput_GVL.xIn_ConnectionRobot[04].5;

// NETWORK 31
END_ACTION

ACTION Input_Safety_active:
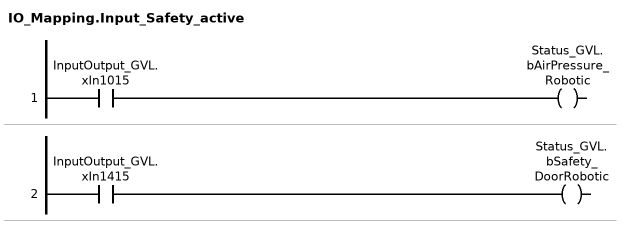
// NETWORK 1
Status_GVL.bAirPressure_Robotic := InputOutput_GVL.xIn1015;

// NETWORK 2
Status_GVL.bSafety_DoorRobotic := InputOutput_GVL.xIn1415;
END_ACTION

ACTION Input_Sensor_active:
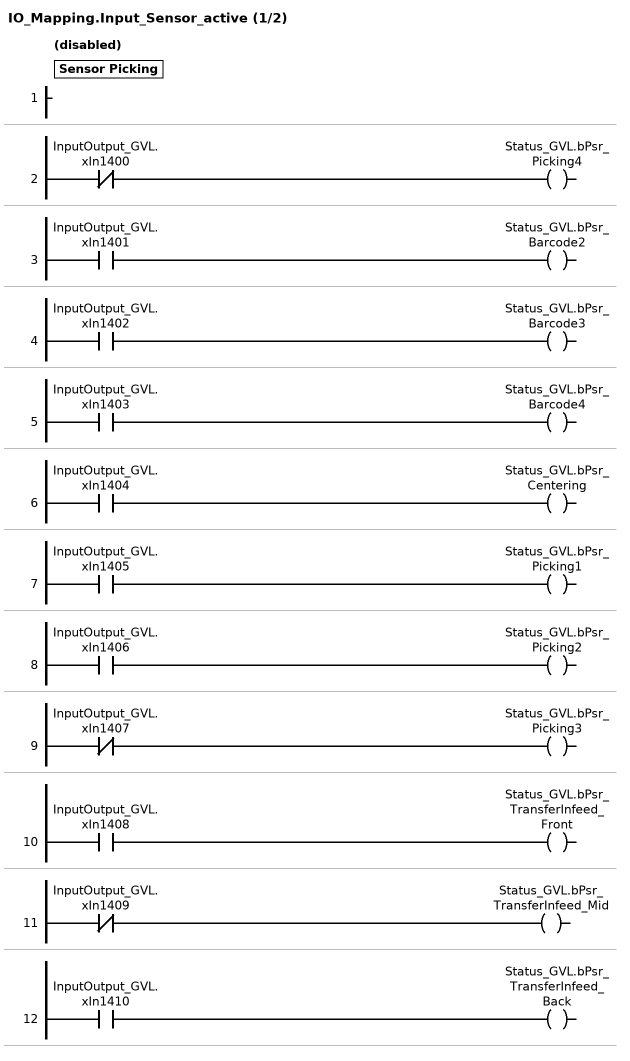
// NETWORK 1 (disabled)
// label: Sensor Picking

// NETWORK 2
Status_GVL.bPsr_Picking4 := NOT InputOutput_GVL.xIn1400;

// NETWORK 3
Status_GVL.bPsr_Barcode2 := InputOutput_GVL.xIn1401;

// NETWORK 4
Status_GVL.bPsr_Barcode3 := InputOutput_GVL.xIn1402;

// NETWORK 5
Status_GVL.bPsr_Barcode4 := InputOutput_GVL.xIn1403;

// NETWORK 6
Status_GVL.bPsr_Centering := InputOutput_GVL.xIn1404;

// NETWORK 7
Status_GVL.bPsr_Picking1 := InputOutput_GVL.xIn1405;

// NETWORK 8
Status_GVL.bPsr_Picking2 := InputOutput_GVL.xIn1406;

// NETWORK 9
Status_GVL.bPsr_Picking3 := NOT InputOutput_GVL.xIn1407;

// NETWORK 10
Status_GVL.bPsr_TransferInfeed_Front := InputOutput_GVL.xIn1408;

// NETWORK 11
Status_GVL.bPsr_TransferInfeed_Mid := NOT InputOutput_GVL.xIn1409;

// NETWORK 12
Status_GVL.bPsr_TransferInfeed_Back := InputOutput_GVL.xIn1410;

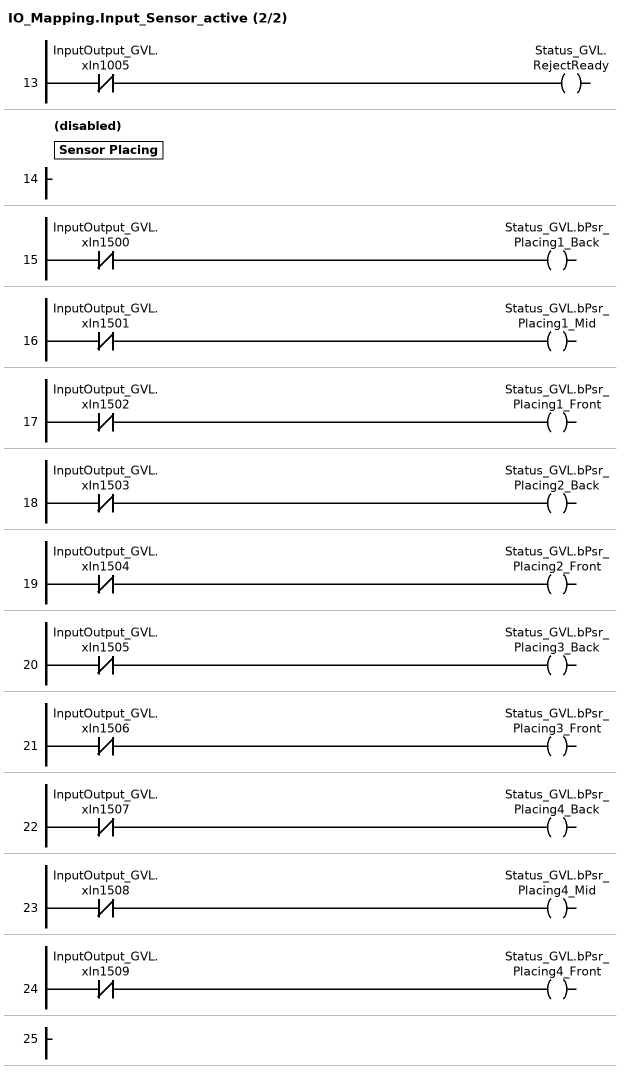
// NETWORK 13
Status_GVL.RejectReady := NOT InputOutput_GVL.xIn1005;

// NETWORK 14 (disabled)
// label: Sensor Placing

// NETWORK 15
Status_GVL.bPsr_Placing1_Back := NOT InputOutput_GVL.xIn1500;

// NETWORK 16
Status_GVL.bPsr_Placing1_Mid := NOT InputOutput_GVL.xIn1501;

// NETWORK 17
Status_GVL.bPsr_Placing1_Front := NOT InputOutput_GVL.xIn1502;

// NETWORK 18
Status_GVL.bPsr_Placing2_Back := NOT InputOutput_GVL.xIn1503;

// NETWORK 19
Status_GVL.bPsr_Placing2_Front := NOT InputOutput_GVL.xIn1504;

// NETWORK 20
Status_GVL.bPsr_Placing3_Back := NOT InputOutput_GVL.xIn1505;

// NETWORK 21
Status_GVL.bPsr_Placing3_Front := NOT InputOutput_GVL.xIn1506;

// NETWORK 22
Status_GVL.bPsr_Placing4_Back := NOT InputOutput_GVL.xIn1507;

// NETWORK 23
Status_GVL.bPsr_Placing4_Mid := NOT InputOutput_GVL.xIn1508;

// NETWORK 24
Status_GVL.bPsr_Placing4_Front := NOT InputOutput_GVL.xIn1509;

// NETWORK 25
END_ACTION

ACTION Output_Indicator_active:
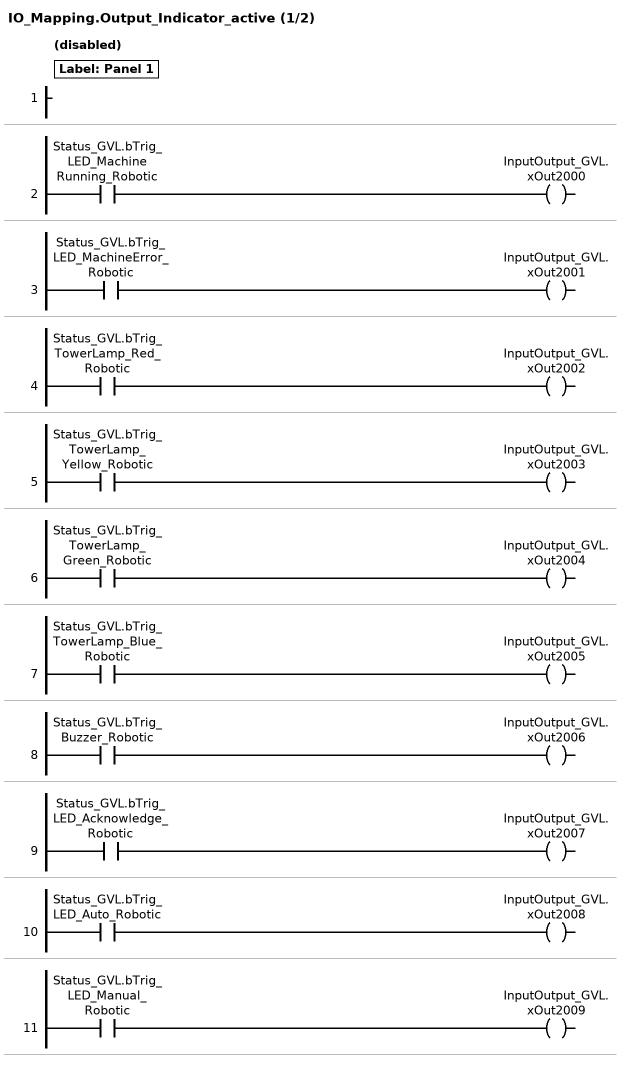
// NETWORK 1 (disabled)
// label: Label: Panel 1

// NETWORK 2
InputOutput_GVL.xOut2000 := Status_GVL.bTrig_LED_MachineRunning_Robotic;

// NETWORK 3
InputOutput_GVL.xOut2001 := Status_GVL.bTrig_LED_MachineError_Robotic;

// NETWORK 4
InputOutput_GVL.xOut2002 := Status_GVL.bTrig_TowerLamp_Red_Robotic;

// NETWORK 5
InputOutput_GVL.xOut2003 := Status_GVL.bTrig_TowerLamp_Yellow_Robotic;

// NETWORK 6
InputOutput_GVL.xOut2004 := Status_GVL.bTrig_TowerLamp_Green_Robotic;

// NETWORK 7
InputOutput_GVL.xOut2005 := Status_GVL.bTrig_TowerLamp_Blue_Robotic;

// NETWORK 8
InputOutput_GVL.xOut2006 := Status_GVL.bTrig_Buzzer_Robotic;

// NETWORK 9
InputOutput_GVL.xOut2007 := Status_GVL.bTrig_LED_Acknowledge_Robotic;

// NETWORK 10
InputOutput_GVL.xOut2008 := Status_GVL.bTrig_LED_Auto_Robotic;

// NETWORK 11
InputOutput_GVL.xOut2009 := Status_GVL.bTrig_LED_Manual_Robotic;

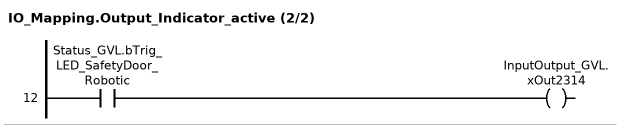
// NETWORK 12
InputOutput_GVL.xOut2314 := Status_GVL.bTrig_LED_SafetyDoor_Robotic;
END_ACTION

ACTION Output_Interlock_active:
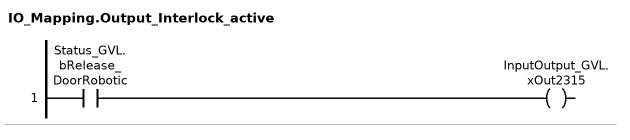
// NETWORK 1
InputOutput_GVL.xOut2315 := Status_GVL.bRelease_DoorRobotic;
END_ACTION

ACTION Output_Motor_active:
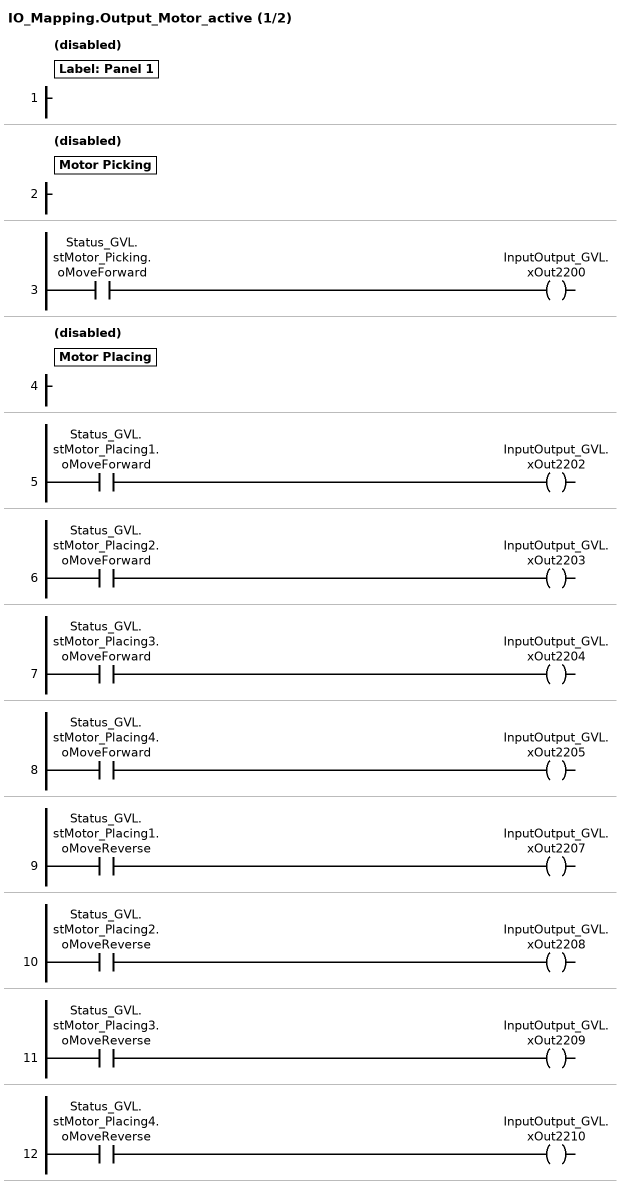
// NETWORK 1 (disabled)
// label: Label: Panel 1

// NETWORK 2 (disabled)
// label: Motor Picking

// NETWORK 3
InputOutput_GVL.xOut2200 := Status_GVL.stMotor_Picking.oMoveForward;

// NETWORK 4 (disabled)
// label: Motor Placing

// NETWORK 5
InputOutput_GVL.xOut2202 := Status_GVL.stMotor_Placing1.oMoveForward;

// NETWORK 6
InputOutput_GVL.xOut2203 := Status_GVL.stMotor_Placing2.oMoveForward;

// NETWORK 7
InputOutput_GVL.xOut2204 := Status_GVL.stMotor_Placing3.oMoveForward;

// NETWORK 8
InputOutput_GVL.xOut2205 := Status_GVL.stMotor_Placing4.oMoveForward;

// NETWORK 9
InputOutput_GVL.xOut2207 := Status_GVL.stMotor_Placing1.oMoveReverse;

// NETWORK 10
InputOutput_GVL.xOut2208 := Status_GVL.stMotor_Placing2.oMoveReverse;

// NETWORK 11
InputOutput_GVL.xOut2209 := Status_GVL.stMotor_Placing3.oMoveReverse;

// NETWORK 12
InputOutput_GVL.xOut2210 := Status_GVL.stMotor_Placing4.oMoveReverse;

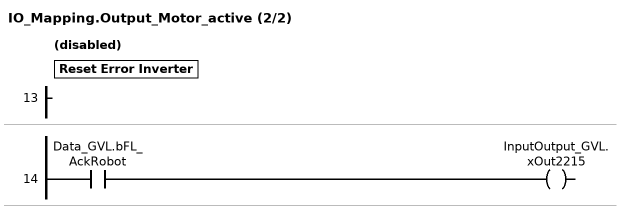
// NETWORK 13 (disabled)
// label: Reset Error Inverter

// NETWORK 14
InputOutput_GVL.xOut2215 := Data_GVL.bFL_AckRobot;
END_ACTION

ACTION Output_Pneumatic_active:
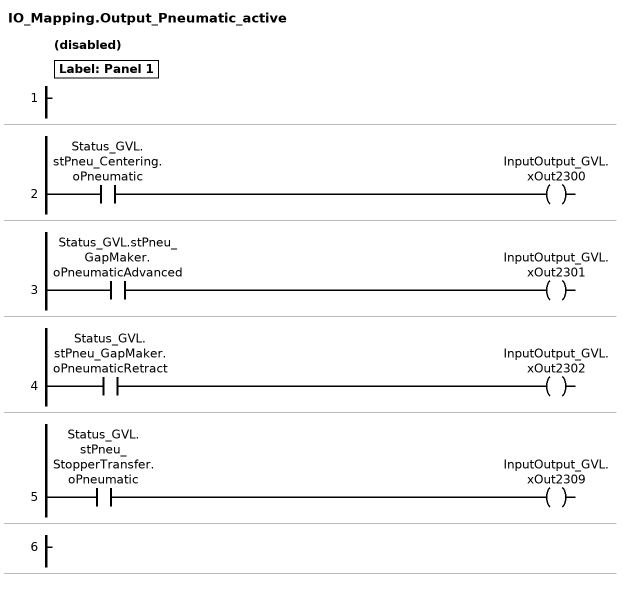
// NETWORK 1 (disabled)
// label: Label: Panel 1

// NETWORK 2
InputOutput_GVL.xOut2300 := Status_GVL.stPneu_Centering.oPneumatic;

// NETWORK 3
InputOutput_GVL.xOut2301 := Status_GVL.stPneu_GapMaker.oPneumaticAdvanced;

// NETWORK 4
InputOutput_GVL.xOut2302 := Status_GVL.stPneu_GapMaker.oPneumaticRetract;

// NETWORK 5
InputOutput_GVL.xOut2309 := Status_GVL.stPneu_StopperTransfer.oPneumatic;

// NETWORK 6
END_ACTION

ACTION Output_Robot_active:
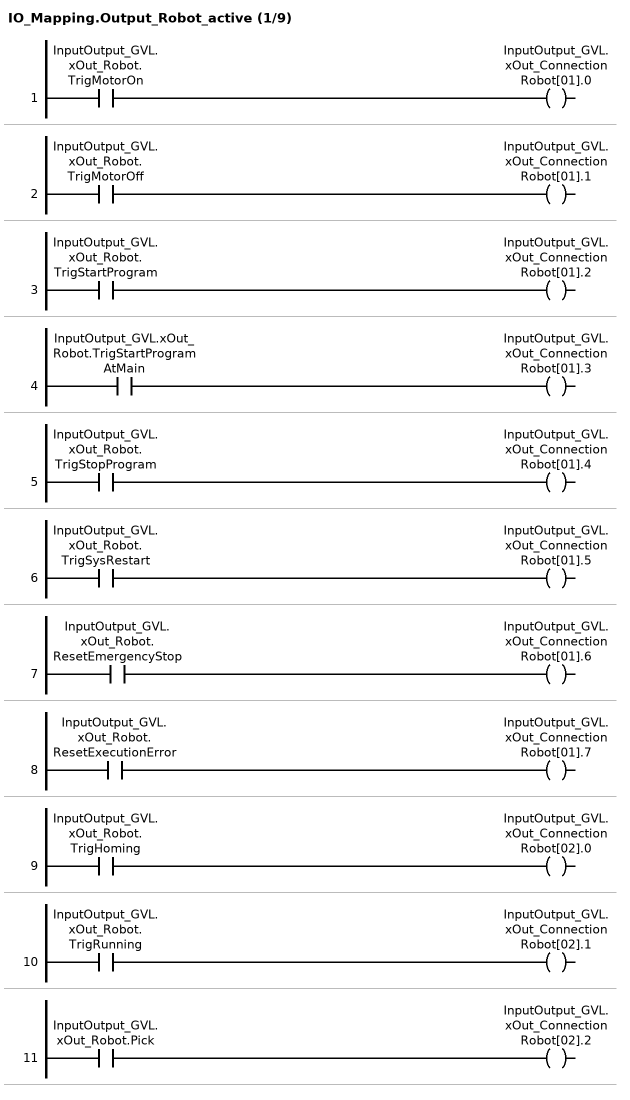
// NETWORK 1
InputOutput_GVL.xOut_ConnectionRobot[01].0 := InputOutput_GVL.xOut_Robot.TrigMotorOn;

// NETWORK 2
InputOutput_GVL.xOut_ConnectionRobot[01].1 := InputOutput_GVL.xOut_Robot.TrigMotorOff;

// NETWORK 3
InputOutput_GVL.xOut_ConnectionRobot[01].2 := InputOutput_GVL.xOut_Robot.TrigStartProgram;

// NETWORK 4
InputOutput_GVL.xOut_ConnectionRobot[01].3 := InputOutput_GVL.xOut_Robot.TrigStartProgramAtMain;

// NETWORK 5
InputOutput_GVL.xOut_ConnectionRobot[01].4 := InputOutput_GVL.xOut_Robot.TrigStopProgram;

// NETWORK 6
InputOutput_GVL.xOut_ConnectionRobot[01].5 := InputOutput_GVL.xOut_Robot.TrigSysRestart;

// NETWORK 7
InputOutput_GVL.xOut_ConnectionRobot[01].6 := InputOutput_GVL.xOut_Robot.ResetEmergencyStop;

// NETWORK 8
InputOutput_GVL.xOut_ConnectionRobot[01].7 := InputOutput_GVL.xOut_Robot.ResetExecutionError;

// NETWORK 9
InputOutput_GVL.xOut_ConnectionRobot[02].0 := InputOutput_GVL.xOut_Robot.TrigHoming;

// NETWORK 10
InputOutput_GVL.xOut_ConnectionRobot[02].1 := InputOutput_GVL.xOut_Robot.TrigRunning;

// NETWORK 11
InputOutput_GVL.xOut_ConnectionRobot[02].2 := InputOutput_GVL.xOut_Robot.Pick;

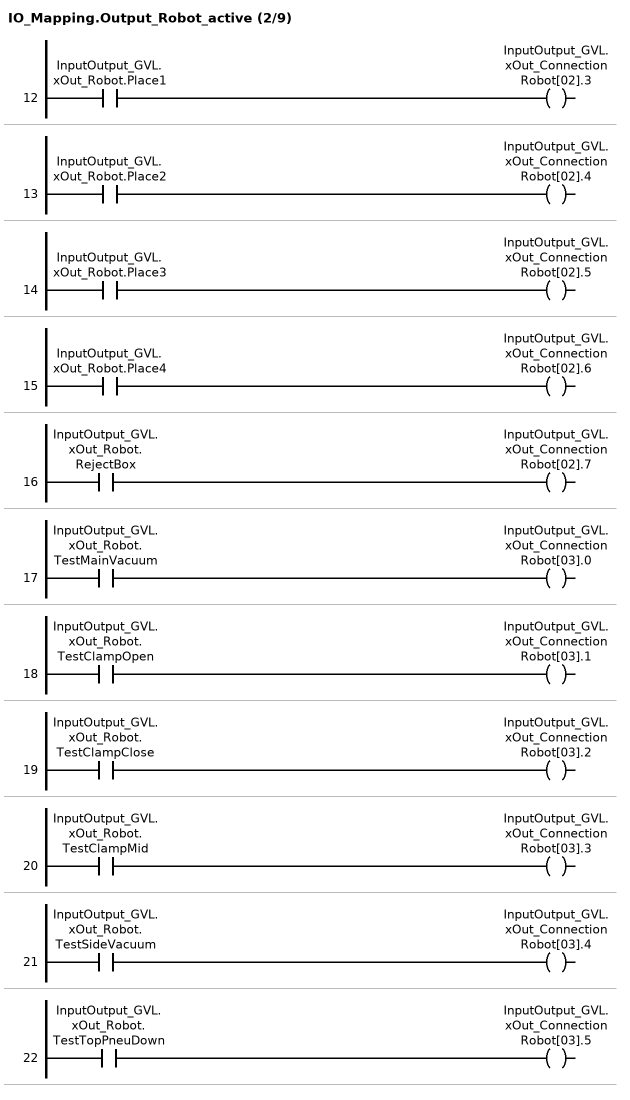
// NETWORK 12
InputOutput_GVL.xOut_ConnectionRobot[02].3 := InputOutput_GVL.xOut_Robot.Place1;

// NETWORK 13
InputOutput_GVL.xOut_ConnectionRobot[02].4 := InputOutput_GVL.xOut_Robot.Place2;

// NETWORK 14
InputOutput_GVL.xOut_ConnectionRobot[02].5 := InputOutput_GVL.xOut_Robot.Place3;

// NETWORK 15
InputOutput_GVL.xOut_ConnectionRobot[02].6 := InputOutput_GVL.xOut_Robot.Place4;

// NETWORK 16
InputOutput_GVL.xOut_ConnectionRobot[02].7 := InputOutput_GVL.xOut_Robot.RejectBox;

// NETWORK 17
InputOutput_GVL.xOut_ConnectionRobot[03].0 := InputOutput_GVL.xOut_Robot.TestMainVacuum;

// NETWORK 18
InputOutput_GVL.xOut_ConnectionRobot[03].1 := InputOutput_GVL.xOut_Robot.TestClampOpen;

// NETWORK 19
InputOutput_GVL.xOut_ConnectionRobot[03].2 := InputOutput_GVL.xOut_Robot.TestClampClose;

// NETWORK 20
InputOutput_GVL.xOut_ConnectionRobot[03].3 := InputOutput_GVL.xOut_Robot.TestClampMid;

// NETWORK 21
InputOutput_GVL.xOut_ConnectionRobot[03].4 := InputOutput_GVL.xOut_Robot.TestSideVacuum;

// NETWORK 22
InputOutput_GVL.xOut_ConnectionRobot[03].5 := InputOutput_GVL.xOut_Robot.TestTopPneuDown;

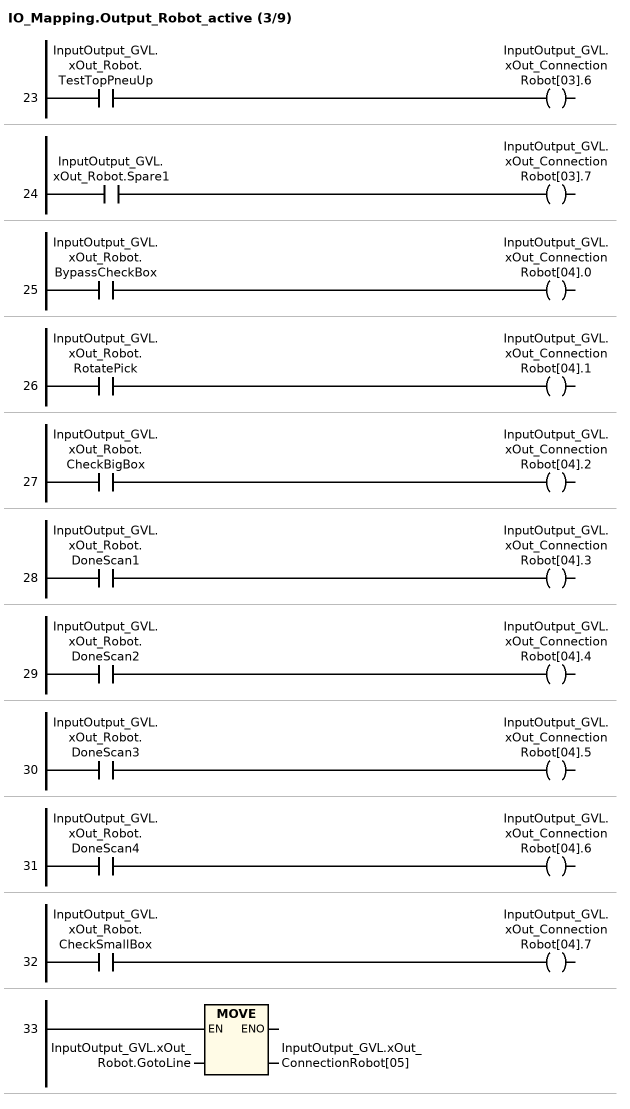
// NETWORK 23
InputOutput_GVL.xOut_ConnectionRobot[03].6 := InputOutput_GVL.xOut_Robot.TestTopPneuUp;

// NETWORK 24
InputOutput_GVL.xOut_ConnectionRobot[03].7 := InputOutput_GVL.xOut_Robot.Spare1;

// NETWORK 25
InputOutput_GVL.xOut_ConnectionRobot[04].0 := InputOutput_GVL.xOut_Robot.BypassCheckBox;

// NETWORK 26
InputOutput_GVL.xOut_ConnectionRobot[04].1 := InputOutput_GVL.xOut_Robot.RotatePick;

// NETWORK 27
InputOutput_GVL.xOut_ConnectionRobot[04].2 := InputOutput_GVL.xOut_Robot.CheckBigBox;

// NETWORK 28
InputOutput_GVL.xOut_ConnectionRobot[04].3 := InputOutput_GVL.xOut_Robot.DoneScan1;

// NETWORK 29
InputOutput_GVL.xOut_ConnectionRobot[04].4 := InputOutput_GVL.xOut_Robot.DoneScan2;

// NETWORK 30
InputOutput_GVL.xOut_ConnectionRobot[04].5 := InputOutput_GVL.xOut_Robot.DoneScan3;

// NETWORK 31
InputOutput_GVL.xOut_ConnectionRobot[04].6 := InputOutput_GVL.xOut_Robot.DoneScan4;

// NETWORK 32
InputOutput_GVL.xOut_ConnectionRobot[04].7 := InputOutput_GVL.xOut_Robot.CheckSmallBox;

// NETWORK 33
InputOutput_GVL.xOut_ConnectionRobot[05] := InputOutput_GVL.xOut_Robot.GotoLine;

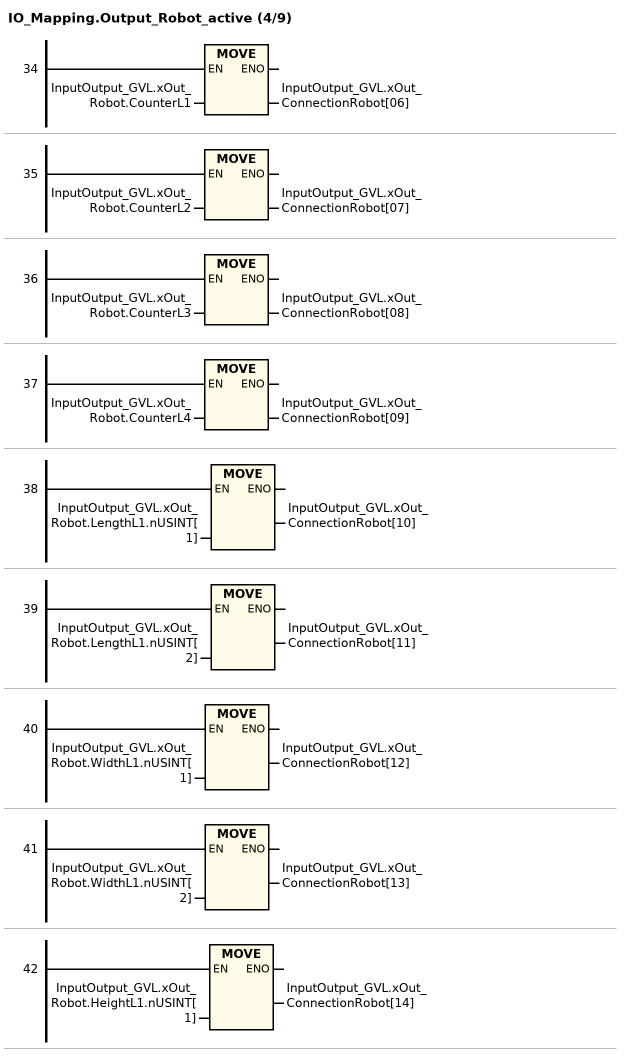
// NETWORK 34
InputOutput_GVL.xOut_ConnectionRobot[06] := InputOutput_GVL.xOut_Robot.CounterL1;

// NETWORK 35
InputOutput_GVL.xOut_ConnectionRobot[07] := InputOutput_GVL.xOut_Robot.CounterL2;

// NETWORK 36
InputOutput_GVL.xOut_ConnectionRobot[08] := InputOutput_GVL.xOut_Robot.CounterL3;

// NETWORK 37
InputOutput_GVL.xOut_ConnectionRobot[09] := InputOutput_GVL.xOut_Robot.CounterL4;

// NETWORK 38
InputOutput_GVL.xOut_ConnectionRobot[10] := InputOutput_GVL.xOut_Robot.LengthL1.nUSINT[1];

// NETWORK 39
InputOutput_GVL.xOut_ConnectionRobot[11] := InputOutput_GVL.xOut_Robot.LengthL1.nUSINT[2];

// NETWORK 40
InputOutput_GVL.xOut_ConnectionRobot[12] := InputOutput_GVL.xOut_Robot.WidthL1.nUSINT[1];

// NETWORK 41
InputOutput_GVL.xOut_ConnectionRobot[13] := InputOutput_GVL.xOut_Robot.WidthL1.nUSINT[2];

// NETWORK 42
InputOutput_GVL.xOut_ConnectionRobot[14] := InputOutput_GVL.xOut_Robot.HeightL1.nUSINT[1];

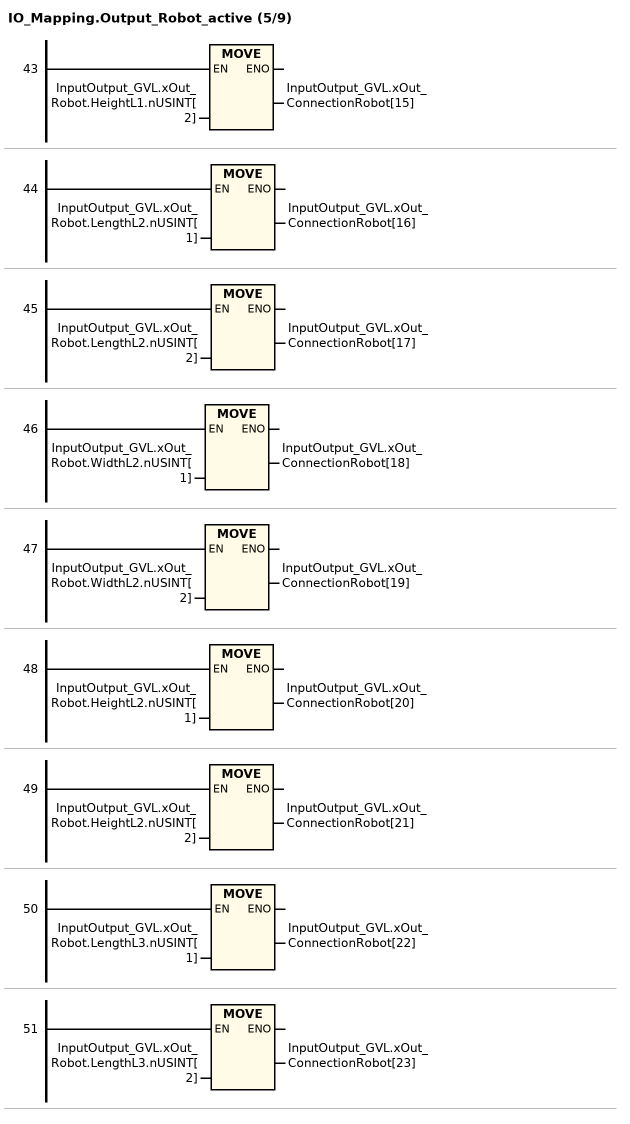
// NETWORK 43
InputOutput_GVL.xOut_ConnectionRobot[15] := InputOutput_GVL.xOut_Robot.HeightL1.nUSINT[2];

// NETWORK 44
InputOutput_GVL.xOut_ConnectionRobot[16] := InputOutput_GVL.xOut_Robot.LengthL2.nUSINT[1];

// NETWORK 45
InputOutput_GVL.xOut_ConnectionRobot[17] := InputOutput_GVL.xOut_Robot.LengthL2.nUSINT[2];

// NETWORK 46
InputOutput_GVL.xOut_ConnectionRobot[18] := InputOutput_GVL.xOut_Robot.WidthL2.nUSINT[1];

// NETWORK 47
InputOutput_GVL.xOut_ConnectionRobot[19] := InputOutput_GVL.xOut_Robot.WidthL2.nUSINT[2];

// NETWORK 48
InputOutput_GVL.xOut_ConnectionRobot[20] := InputOutput_GVL.xOut_Robot.HeightL2.nUSINT[1];

// NETWORK 49
InputOutput_GVL.xOut_ConnectionRobot[21] := InputOutput_GVL.xOut_Robot.HeightL2.nUSINT[2];

// NETWORK 50
InputOutput_GVL.xOut_ConnectionRobot[22] := InputOutput_GVL.xOut_Robot.LengthL3.nUSINT[1];

// NETWORK 51
InputOutput_GVL.xOut_ConnectionRobot[23] := InputOutput_GVL.xOut_Robot.LengthL3.nUSINT[2];

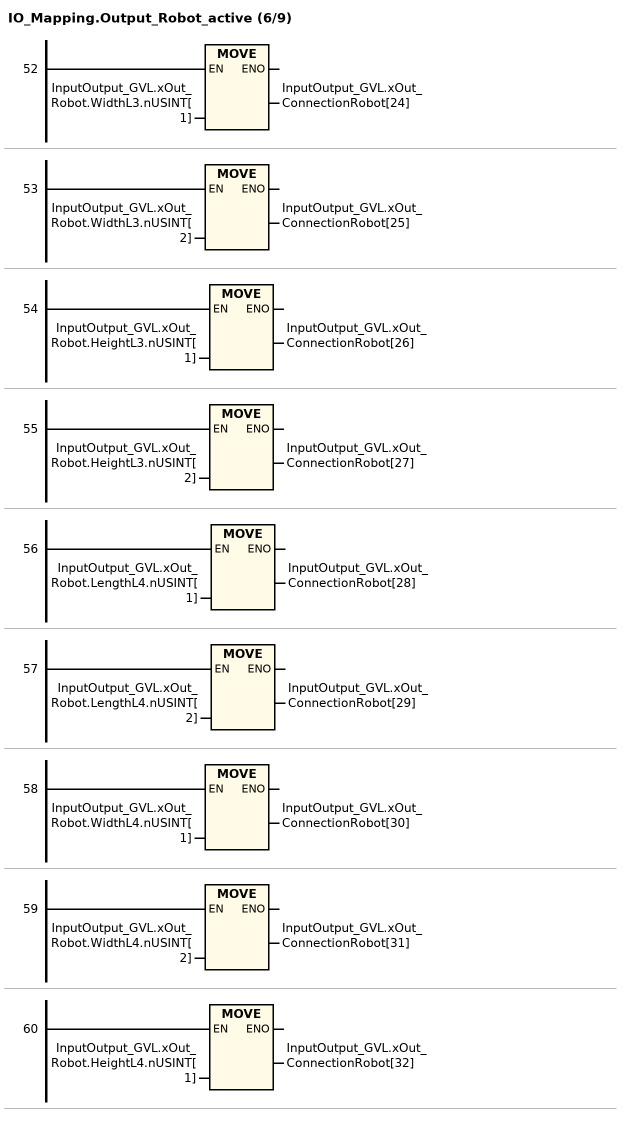
// NETWORK 52
InputOutput_GVL.xOut_ConnectionRobot[24] := InputOutput_GVL.xOut_Robot.WidthL3.nUSINT[1];

// NETWORK 53
InputOutput_GVL.xOut_ConnectionRobot[25] := InputOutput_GVL.xOut_Robot.WidthL3.nUSINT[2];

// NETWORK 54
InputOutput_GVL.xOut_ConnectionRobot[26] := InputOutput_GVL.xOut_Robot.HeightL3.nUSINT[1];

// NETWORK 55
InputOutput_GVL.xOut_ConnectionRobot[27] := InputOutput_GVL.xOut_Robot.HeightL3.nUSINT[2];

// NETWORK 56
InputOutput_GVL.xOut_ConnectionRobot[28] := InputOutput_GVL.xOut_Robot.LengthL4.nUSINT[1];

// NETWORK 57
InputOutput_GVL.xOut_ConnectionRobot[29] := InputOutput_GVL.xOut_Robot.LengthL4.nUSINT[2];

// NETWORK 58
InputOutput_GVL.xOut_ConnectionRobot[30] := InputOutput_GVL.xOut_Robot.WidthL4.nUSINT[1];

// NETWORK 59
InputOutput_GVL.xOut_ConnectionRobot[31] := InputOutput_GVL.xOut_Robot.WidthL4.nUSINT[2];

// NETWORK 60
InputOutput_GVL.xOut_ConnectionRobot[32] := InputOutput_GVL.xOut_Robot.HeightL4.nUSINT[1];

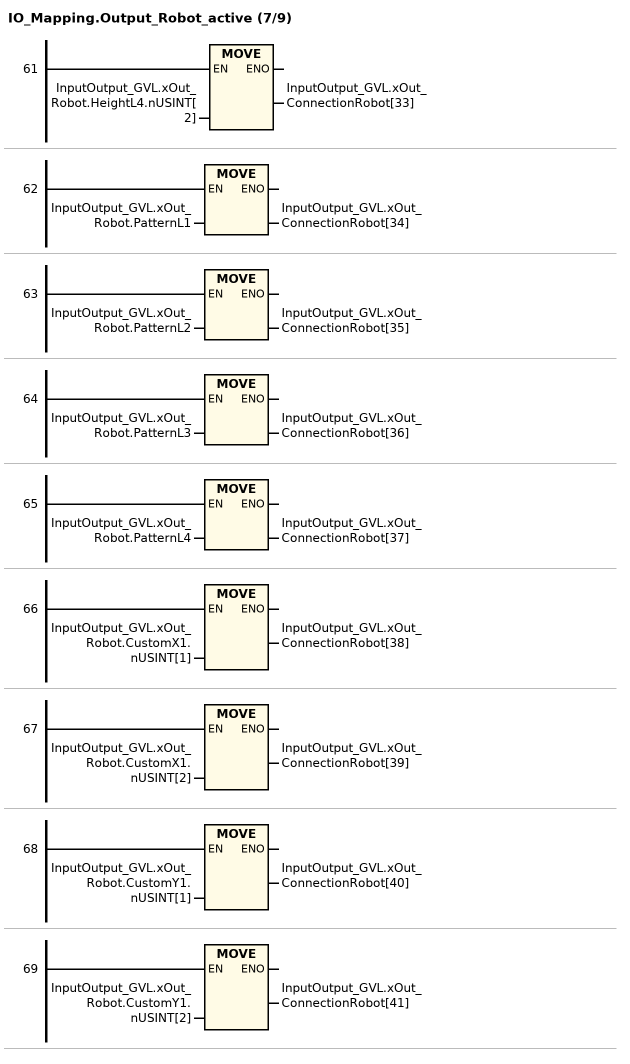
// NETWORK 61
InputOutput_GVL.xOut_ConnectionRobot[33] := InputOutput_GVL.xOut_Robot.HeightL4.nUSINT[2];

// NETWORK 62
InputOutput_GVL.xOut_ConnectionRobot[34] := InputOutput_GVL.xOut_Robot.PatternL1;

// NETWORK 63
InputOutput_GVL.xOut_ConnectionRobot[35] := InputOutput_GVL.xOut_Robot.PatternL2;

// NETWORK 64
InputOutput_GVL.xOut_ConnectionRobot[36] := InputOutput_GVL.xOut_Robot.PatternL3;

// NETWORK 65
InputOutput_GVL.xOut_ConnectionRobot[37] := InputOutput_GVL.xOut_Robot.PatternL4;

// NETWORK 66
InputOutput_GVL.xOut_ConnectionRobot[38] := InputOutput_GVL.xOut_Robot.CustomX1.nUSINT[1];

// NETWORK 67
InputOutput_GVL.xOut_ConnectionRobot[39] := InputOutput_GVL.xOut_Robot.CustomX1.nUSINT[2];

// NETWORK 68
InputOutput_GVL.xOut_ConnectionRobot[40] := InputOutput_GVL.xOut_Robot.CustomY1.nUSINT[1];

// NETWORK 69
InputOutput_GVL.xOut_ConnectionRobot[41] := InputOutput_GVL.xOut_Robot.CustomY1.nUSINT[2];

